LIN {X 0,Y 305.398,Z 312.447,A -85,B 0,C 180,E1 -15799.883,E2 -15799.883} C_VEL
LIN {X 0,Y 305.449,Z 312.421,A -85,B 0,C 180,E1 -15803.636,E2 -15803.636} C_VEL
LIN {X 0,Y 305.452,Z 312.437,A -85,B 0,C 180,E1 -15806.482,E2 -15806.482} C_VEL
LIN {X 0,Y 305.417,Z 312.439,A -85,B 0,C 180,E1 -15809.586,E2 -15809.586} C_VEL
LIN {X 0,Y 305.444,Z 312.436,A -85,B 0,C 180,E1 -15812.601,E2 -15812.601} C_VEL
LIN {X 0,Y 305.461,Z 312.428,A -85,B 0,C 180,E1 -15815.535,E2 -15815.535} C_VEL
LIN {X 0,Y 305.498,Z 312.423,A -85,B 0,C 180,E1 -15819.814,E2 -15819.814} C_VEL
LIN {X 0,Y 305.56,Z 312.415,A -85,B 0,C 180,E1 -15822.602,E2 -15822.602} C_VEL
LIN {X 0,Y 305.635,Z 312.412,A -85,B 0,C 180,E1 -15825.349,E2 -15825.349} C_VEL
LIN {X 0,Y 305.622,Z 312.411,A -85,B 0,C 180,E1 -15829.399,E2 -15829.399} C_VEL
LIN {X 0,Y 305.737,Z 312.393,A -85,B 0,C 180,E1 -15832.073,E2 -15832.073} C_VEL
LIN {X 0,Y 305.66,Z 312.409,A -85,B 0,C 180,E1 -15834.723,E2 -15834.723} C_VEL
LIN {X 0,Y 305.943,Z 312.363,A -85,B 0,C 180,E1 -15838.684,E2 -15838.684} C_VEL
LIN {X 0,Y 305.945,Z 312.371,A -85,B 0,C 180,E1 -15841.317,E2 -15841.317} C_VEL
LIN {X 0,Y 305.838,Z 312.386,A -85,B 0,C 180,E1 -15846.598,E2 -15846.598} C_VEL
LIN {X 0,Y 305.723,Z 312.392,A -85,B 0,C 180,E1 -15849.26,E2 -15849.26} C_VEL
LIN {X 0,Y 305.576,Z 312.407,A -85,B 0,C 180,E1 -15853.297,E2 -15853.297} C_VEL
LIN {X 0,Y 305.581,Z 312.419,A -85,B 0,C 180,E1 -15856.021,E2 -15856.021} C_VEL
LIN {X 0,Y 305.565,Z 312.413,A -85,B 0,C 180,E1 -15859.446,E2 -15859.446} C_VEL
LIN {X 0,Y 305.478,Z 312.424,A -85,B 0,C 180,E1 -15863.042,E2 -15863.042} C_VEL
LIN {X 0,Y 305.543,Z 312.424,A -85,B 0,C 180,E1 -15866.231,E2 -15866.231} C_VEL
LIN {X 0,Y 305.485,Z 312.426,A -85,B 0,C 180,E1 -15869.052,E2 -15869.052} C_VEL
LIN {X 0,Y 305.437,Z 312.43,A -85,B 0,C 180,E1 -15871.953,E2 -15871.953} C_VEL
LIN {X 0,Y 305.453,Z 312.435,A -85,B 0,C 180,E1 -15875.115,E2 -15875.115} C_VEL
LIN {X 0,Y 305.483,Z 312.433,A -85,B 0,C 180,E1 -15878.541,E2 -15878.541} C_VEL
LIN {X 0,Y 305.49,Z 312.429,A -85,B 0,C 180,E1 -15882.597,E2 -15882.597} C_VEL
LIN {X 0,Y 305.485,Z 312.416,A -85,B 0,C 180,E1 -15886.359,E2 -15886.359} C_VEL
LIN {X 0,Y 305.494,Z 312.42,A -85,B 0,C 180,E1 -15889.901,E2 -15889.901} C_VEL
LIN {X 0,Y 305.495,Z 312.51,A -85,B 0,C 180,E1 -15893.574,E2 -15893.574} C_VEL
LIN {X 0,Y 308.431,Z 323.615,A -85,B 0,C 180,E1 -15897.469,E2 -15897.469} C_VEL
LIN {X 0,Y 310.794,Z 334.247,A -85,B 0,C 180,E1 -15900.913,E2 -15900.913} C_VEL
LIN {X 0,Y 311.289,Z 336.675,A -85,B 0,C 180,E1 -15901.649,E2 -15901.649} C_VEL
LIN {X 0,Y 314.76,Z 344.965,A -85,B 0,C 180,E1 -15902.279,E2 -15902.279} C_VEL
LIN {X 0,Y 319.961,Z 370.288,A -85,B 0,C 180,E1 -15903.522,E2 -15903.522} C_VEL
LIN {X 0,Y 321.701,Z 382.338,A -85,B 0,C 180,E1 -15904.017,E2 -15904.017} C_VEL
LIN {X 0,Y 319.792,Z 446.05,A -85,B 0,C 180,E1 -15905.495,E2 -15905.495} C_VEL
LIN {X 0,Y 318.807,Z 458.991,A -85,B 0,C 180,E1 -15906.02,E2 -15906.02} C_VEL
LIN {X 0,Y 317.343,Z 471.558,A -85,B 0,C 180,E1 -15906.769,E2 -15906.769} C_VEL
LIN {X 0,Y 315.685,Z 483.551,A -85,B 0,C 180,E1 -15907.764,E2 -15907.764} C_VEL
LIN {X 0,Y 313.762,Z 495.004,A -85,B 0,C 180,E1 -15909.001,E2 -15909.001} C_VEL
LIN {X 0,Y 311.866,Z 505.349,A -85,B 0,C 180,E1 -15910.417,E2 -15910.417} C_VEL
LIN {X 0,Y 310.092,Z 513.837,A -85,B 0,C 180,E1 -15911.845,E2 -15911.845} C_VEL
LIN {X 0,Y 308.629,Z 521.845,A -85,B 0,C 180,E1 -15913.503,E2 -15913.503} C_VEL
LIN {X 0,Y 307.051,Z 529.381,A -85,B 0,C 180,E1 -15915.42,E2 -15915.42} C_VEL
LIN {X 0,Y 305.65,Z 535.589,A -85,B 0,C 180,E1 -15917.385,E2 -15917.385} C_VEL
LIN {X 0,Y 304.733,Z 540.548,A -85,B 0,C 180,E1 -15919.37,E2 -15919.37} C_VEL
LIN {X 0,Y 304.146,Z 544.402,A -85,B 0,C 180,E1 -15921.364,E2 -15921.364} C_VEL
LIN {X 0,Y 303.744,Z 547.251,A -85,B 0,C 180,E1 -15923.359,E2 -15923.359} C_VEL
LIN {X 0,Y 303.632,Z 549.583,A -85,B 0,C 180,E1 -15926.02,E2 -15926.02} C_VEL
LIN {X 0,Y 303.623,Z 550.168,A -85,B 0,C 180,E1 -15927.349,E2 -15927.349} C_VEL
LIN {X 0,Y 303.607,Z 550.324,A -85,B 0,C 180,E1 -15928.676,E2 -15928.676} C_VEL
LIN {X 0,Y 303.67,Z 550.08,A -85,B 0,C 180,E1 -15930.002,E2 -15930.002} C_VEL
LIN {X 0,Y 303.636,Z 549.443,A -85,B 0,C 180,E1 -15931.328,E2 -15931.328} C_VEL
LIN {X 0,Y 303.646,Z 548.413,A -85,B 0,C 180,E1 -15932.655,E2 -15932.655} C_VEL
LIN {X 0,Y 303.671,Z 546.934,A -85,B 0,C 180,E1 -15933.983,E2 -15933.983} C_VEL
LIN {X 0,Y 303.732,Z 544.307,A -85,B 0,C 180,E1 -15935.746,E2 -15935.746} C_VEL
LIN {X 0,Y 303.942,Z 539.784,A -85,B 0,C 180,E1 -15937.977,E2 -15937.977} C_VEL
LIN {X 0,Y 304.442,Z 533.453,A -85,B 0,C 180,E1 -15940.308,E2 -15940.308} C_VEL
LIN {X 0,Y 305.118,Z 526.541,A -85,B 0,C 180,E1 -15942.304,E2 -15942.304} C_VEL
LIN {X 0,Y 305.993,Z 519.484,A -85,B 0,C 180,E1 -15943.957,E2 -15943.957} C_VEL
LIN {X 0,Y 307.039,Z 510.967,A -85,B 0,C 180,E1 -15945.604,E2 -15945.604} C_VEL
LIN {X 0,Y 308.259,Z 500.414,A -85,B 0,C 180,E1 -15947.243,E2 -15947.243} C_VEL
LIN {X 0,Y 309.206,Z 491.39,A -85,B 0,C 180,E1 -15948.385,E2 -15948.385} C_VEL
LIN {X 0,Y 310.42,Z 480.275,A -85,B 0,C 180,E1 -15949.51,E2 -15949.51} C_VEL
LIN {X 0,Y 311.558,Z 467.945,A -85,B 0,C 180,E1 -15950.467,E2 -15950.467} C_VEL
LIN {X 0,Y 312.492,Z 454.939,A -85,B 0,C 180,E1 -15951.179,E2 -15951.179} C_VEL
LIN {X 0,Y 313.069,Z 441.053,A -85,B 0,C 180,E1 -15951.656,E2 -15951.656} C_VEL
LIN {X 0,Y 314.281,Z 379.106,A -85,B 0,C 180,E1 -15953.068,E2 -15953.068} C_VEL
LIN {X 0,Y 308.709,Z 337.55,A -85,B 0,C 180,E1 -15954.454,E2 -15954.454} C_VEL
LIN {X 0,Y 309.301,Z 331.86,A -85,B 0,C 180,E1 -15955.94,E2 -15955.94} C_VEL
LIN {X 0,Y 307.601,Z 322.197,A -85,B 0,C 180,E1 -15958.674,E2 -15958.674} C_VEL
LIN {X 0,Y 305.475,Z 312.435,A -85,B 0,C 180,E1 -15961.581,E2 -15961.581} C_VEL
LIN {X 0,Y 305.469,Z 312.433,A -85,B 0,C 180,E1 -15965.114,E2 -15965.114} C_VEL
LIN {X 0,Y 305.456,Z 312.438,A -85,B 0,C 180,E1 -15968.53,E2 -15968.53} C_VEL
LIN {X 0,Y 305.462,Z 312.438,A -85,B 0,C 180,E1 -15972.587,E2 -15972.587} C_VEL
LIN {X 0,Y 305.432,Z 312.439,A -85,B 0,C 180,E1 -15976.346,E2 -15976.346} C_VEL
LIN {X 0,Y 305.465,Z 312.431,A -85,B 0,C 180,E1 -15979.893,E2 -15979.893} C_VEL
LIN {X 0,Y 305.487,Z 312.429,A -85,B 0,C 180,E1 -15983.632,E2 -15983.632} C_VEL
LIN {X 0,Y 305.472,Z 312.431,A -85,B 0,C 180,E1 -15986.484,E2 -15986.484} C_VEL
LIN {X 0,Y 305.503,Z 312.429,A -85,B 0,C 180,E1 -15990.951,E2 -15990.951} C_VEL
LIN {X 0,Y 305.579,Z 312.418,A -85,B 0,C 180,E1 -15994.088,E2 -15994.088} C_VEL
LIN {X 0,Y 305.481,Z 312.429,A -85,B 0,C 180,E1 -15998.401,E2 -15998.401} C_VEL
LIN {X 0,Y 305.525,Z 312.424,A -85,B 0,C 180,E1 -16001.213,E2 -16001.213} C_VEL
LIN {X 0,Y 305.633,Z 312.412,A -85,B 0,C 180,E1 -16005.348,E2 -16005.348} C_VEL
LIN {X 0,Y 305.642,Z 312.412,A -85,B 0,C 180,E1 -16009.4,E2 -16009.4} C_VEL
LIN {X 0,Y 305.754,Z 312.392,A -85,B 0,C 180,E1 -16012.072,E2 -16012.072} C_VEL
LIN {X 0,Y 305.677,Z 312.401,A -85,B 0,C 180,E1 -16014.723,E2 -16014.723} C_VEL
LIN {X 0,Y 305.96,Z 312.37,A -85,B 0,C 180,E1 -16018.683,E2 -16018.683} C_VEL
LIN {X 0,Y 305.96,Z 312.369,A -85,B 0,C 180,E1 -16021.316,E2 -16021.316} C_VEL
LIN {X 0,Y 305.687,Z 312.396,A -85,B 0,C 180,E1 -16025.276,E2 -16025.276} C_VEL
LIN {X 0,Y 305.778,Z 312.389,A -85,B 0,C 180,E1 -16027.926,E2 -16027.926} C_VEL
LIN {X 0,Y 305.605,Z 312.415,A -85,B 0,C 180,E1 -16031.945,E2 -16031.945} C_VEL
LIN {X 0,Y 305.615,Z 312.413,A -85,B 0,C 180,E1 -16035.014,E2 -16035.014} C_VEL
LIN {X 0,Y 305.524,Z 312.43,A -85,B 0,C 180,E1 -16038.786,E2 -16038.786} C_VEL
LIN {X 0,Y 305.492,Z 312.432,A -85,B 0,C 180,E1 -16043.039,E2 -16043.039} C_VEL
LIN {X 0,Y 305.532,Z 312.423,A -85,B 0,C 180,E1 -16046.218,E2 -16046.218} C_VEL
LIN {X 0,Y 305.494,Z 312.431,A -85,B 0,C 180,E1 -16049.047,E2 -16049.047} C_VEL
LIN {X 0,Y 305.448,Z 312.433,A -85,B 0,C 180,E1 -16051.951,E2 -16051.951} C_VEL
LIN {X 0,Y 305.468,Z 312.434,A -85,B 0,C 180,E1 -16055.112,E2 -16055.112} C_VEL
LIN {X 0,Y 305.445,Z 312.433,A -85,B 0,C 180,E1 -16058.525,E2 -16058.525} C_VEL
LIN {X 0,Y 305.478,Z 312.429,A -85,B 0,C 180,E1 -16062.588,E2 -16062.588} C_VEL
LIN {X 0,Y 305.459,Z 312.435,A -85,B 0,C 180,E1 -16067.413,E2 -16067.413} C_VEL
LIN {X 0,Y 305.499,Z 312.43,A -85,B 0,C 180,E1 -16071.599,E2 -16071.599} C_VEL
LIN {X 0,Y 305.466,Z 312.431,A -85,B 0,C 180,E1 -16074.885,E2 -16074.885} C_VEL
LIN {X 0,Y 305.453,Z 312.435,A -85,B 0,C 180,E1 -16078.354,E2 -16078.354} C_VEL
LIN {X 0,Y 305.516,Z 312.425,A -85,B 0,C 180,E1 -16081.112,E2 -16081.112} C_VEL
LIN {X 0,Y 305.574,Z 312.423,A -85,B 0,C 180,E1 -16084.086,E2 -16084.086} C_VEL
LIN {X 0,Y 305.532,Z 312.428,A -85,B 0,C 180,E1 -16088.403,E2 -16088.403} C_VEL
LIN {X 0,Y 305.595,Z 312.416,A -85,B 0,C 180,E1 -16091.216,E2 -16091.216} C_VEL
LIN {X 0,Y 305.651,Z 312.41,A -85,B 0,C 180,E1 -16095.347,E2 -16095.347} C_VEL
LIN {X 0,Y 305.665,Z 312.589,A -85,B 0,C 180,E1 -16099.231,E2 -16099.231} C_VEL
LIN {X 0,Y 306.522,Z 316.593,A -85,B 0,C 180,E1 -16100.487,E2 -16100.487} C_VEL
LIN {X 0,Y 312.904,Z 335.521,A -85,B 0,C 180,E1 -16101.395,E2 -16101.395} C_VEL
LIN {X 0,Y 314.899,Z 346.476,A -85,B 0,C 180,E1 -16101.787,E2 -16101.787} C_VEL
LIN {X 0,Y 313.086,Z 424.785,A -85,B 0,C 180,E1 -16103.594,E2 -16103.594} C_VEL
LIN {X 0,Y 312.418,Z 438.468,A -85,B 0,C 180,E1 -16104.188,E2 -16104.188} C_VEL
LIN {X 0,Y 311.682,Z 450.742,A -85,B 0,C 180,E1 -16104.985,E2 -16104.985} C_VEL
LIN {X 0,Y 310.637,Z 463.358,A -85,B 0,C 180,E1 -16106.106,E2 -16106.106} C_VEL
LIN {X 0,Y 309.466,Z 474.611,A -85,B 0,C 180,E1 -16107.395,E2 -16107.395} C_VEL
LIN {X 0,Y 308.216,Z 484.757,A -85,B 0,C 180,E1 -16108.855,E2 -16108.855} C_VEL
LIN {X 0,Y 306.982,Z 494.708,A -85,B 0,C 180,E1 -16110.654,E2 -16110.654} C_VEL
LIN {X 0,Y 305.871,Z 503.471,A -85,B 0,C 180,E1 -16112.632,E2 -16112.632} C_VEL
LIN {X 0,Y 305.06,Z 510.446,A -85,B 0,C 180,E1 -16114.623,E2 -16114.623} C_VEL
LIN {X 0,Y 304.552,Z 516.023,A -85,B 0,C 180,E1 -16116.624,E2 -16116.624} C_VEL
LIN {X 0,Y 304.078,Z 520.42,A -85,B 0,C 180,E1 -16118.638,E2 -16118.638} C_VEL
LIN {X 0,Y 303.697,Z 523.738,A -85,B 0,C 180,E1 -16120.667,E2 -16120.667} C_VEL
LIN {X 0,Y 303.593,Z 525.384,A -85,B 0,C 180,E1 -16122.023,E2 -16122.023} C_VEL
LIN {X 0,Y 303.543,Z 526.681,A -85,B 0,C 180,E1 -16123.485,E2 -16123.485} C_VEL
LIN {X 0,Y 303.461,Z 527.755,A -85,B 0,C 180,E1 -16126.133,E2 -16126.133} C_VEL
LIN {X 0,Y 303.688,Z 527.448,A -85,B 0,C 180,E1 -16128.409,E2 -16128.409} C_VEL
LIN {X 0,Y 303.99,Z 526.316,A -85,B 0,C 180,E1 -16130.289,E2 -16130.289} C_VEL
LIN {X 0,Y 304.616,Z 523.753,A -85,B 0,C 180,E1 -16132.652,E2 -16132.652} C_VEL
LIN {X 0,Y 305.608,Z 519.497,A -85,B 0,C 180,E1 -16135.176,E2 -16135.176} C_VEL
LIN {X 0,Y 306.708,Z 514.599,A -85,B 0,C 180,E1 -16137.274,E2 -16137.274} C_VEL
LIN {X 0,Y 308.159,Z 508.31,A -85,B 0,C 180,E1 -16139.36,E2 -16139.36} C_VEL
LIN {X 0,Y 309.903,Z 500.374,A -85,B 0,C 180,E1 -16141.437,E2 -16141.437} C_VEL
LIN {X 0,Y 311.708,Z 491.871,A -85,B 0,C 180,E1 -16143.192,E2 -16143.192} C_VEL
LIN {X 0,Y 313.595,Z 481.907,A -85,B 0,C 180,E1 -16144.851,E2 -16144.851} C_VEL
LIN {X 0,Y 315.375,Z 471.812,A -85,B 0,C 180,E1 -16146.192,E2 -16146.192} C_VEL
LIN {X 0,Y 316.932,Z 461.289,A -85,B 0,C 180,E1 -16147.313,E2 -16147.313} C_VEL
LIN {X 0,Y 318.315,Z 449.539,A -85,B 0,C 180,E1 -16148.283,E2 -16148.283} C_VEL
LIN {X 0,Y 319.552,Z 436.467,A -85,B 0,C 180,E1 -16149.065,E2 -16149.065} C_VEL
LIN {X 0,Y 320.342,Z 423.599,A -85,B 0,C 180,E1 -16149.575,E2 -16149.575} C_VEL
LIN {X 0,Y 322.577,Z 350.795,A -85,B 0,C 180,E1 -16151.238,E2 -16151.238} C_VEL
LIN {X 0,Y 316.186,Z 336.137,A -85,B 0,C 180,E1 -16152.328,E2 -16152.328} C_VEL
LIN {X 0,Y 308.719,Z 321.185,A -85,B 0,C 180,E1 -16153.627,E2 -16153.627} C_VEL
LIN {X 0,Y 306.652,Z 317.269,A -85,B 0,C 180,E1 -16154.031,E2 -16154.031} C_VEL
LIN {X 0,Y 305.411,Z 312.433,A -85,B 0,C 180,E1 -16155.821,E2 -16155.821} C_VEL
LIN {X 0,Y 305.404,Z 312.433,A -85,B 0,C 180,E1 -16156.566,E2 -16156.566} C_VEL
LIN {X 0,Y 304.731,Z 312.527,A -85,B 0,C 180,E1 -16157.666,E2 -16157.666} C_VEL
LIN {X 0,Y 301.878,Z 312.895,A -85,B 0,C 180,E1 -16159.458,E2 -16159.458} C_VEL
LIN {X 0,Y 299.471,Z 313.197,A -85,B 0,C 180,E1 -16160.912,E2 -16160.912} C_VEL
LIN {X 0,Y 298.452,Z 313.314,A -85,B 0,C 180,E1 -16162.038,E2 -16162.038} C_VEL
LIN {X 0,Y 298.375,Z 313.318,A -85,B 0,C 180,E1 -16162.419,E2 -16162.419} C_VEL
LIN {X 0,Y 298.395,Z 313.301,A -85,B 0,C 180,E1 -16165.58,E2 -16165.58} C_VEL
LIN {X 0,Y 298.364,Z 313.313,A -85,B 0,C 180,E1 -16168.788,E2 -16168.788} C_VEL
LIN {X 0,Y 298.4,Z 313.309,A -85,B 0,C 180,E1 -16171.898,E2 -16171.898} C_VEL
LIN {X 0,Y 298.426,Z 313.304,A -85,B 0,C 180,E1 -16174.919,E2 -16174.919} C_VEL
LIN {X 0,Y 298.426,Z 313.301,A -85,B 0,C 180,E1 -16179.314,E2 -16179.314} C_VEL
LIN {X 0,Y 298.524,Z 313.295,A -85,B 0,C 180,E1 -16182.179,E2 -16182.179} C_VEL
LIN {X 0,Y 298.58,Z 313.291,A -85,B 0,C 180,E1 -16184.994,E2 -16184.994} C_VEL
LIN {X 0,Y 298.578,Z 313.288,A -85,B 0,C 180,E1 -16189.146,E2 -16189.146} C_VEL
LIN {X 0,Y 298.688,Z 313.273,A -85,B 0,C 180,E1 -16191.884,E2 -16191.884} C_VEL
LIN {X 0,Y 298.629,Z 313.283,A -85,B 0,C 180,E1 -16194.599,E2 -16194.599} C_VEL
LIN {X 0,Y 298.91,Z 313.239,A -85,B 0,C 180,E1 -16198.653,E2 -16198.653} C_VEL
LIN {X 0,Y 298.911,Z 313.248,A -85,B 0,C 180,E1 -16201.348,E2 -16201.348} C_VEL
LIN {X 0,Y 298.784,Z 313.263,A -85,B 0,C 180,E1 -16206.754,E2 -16206.754} C_VEL
LIN {X 0,Y 298.668,Z 313.272,A -85,B 0,C 180,E1 -16209.481,E2 -16209.481} C_VEL
LIN {X 0,Y 298.539,Z 313.282,A -85,B 0,C 180,E1 -16213.616,E2 -16213.616} C_VEL
LIN {X 0,Y 298.536,Z 313.298,A -85,B 0,C 180,E1 -16216.41,E2 -16216.41} C_VEL
LIN {X 0,Y 298.5,Z 313.295,A -85,B 0,C 180,E1 -16219.656,E2 -16219.656} C_VEL
LIN {X 0,Y 298.446,Z 313.298,A -85,B 0,C 180,E1 -16223.599,E2 -16223.599} C_VEL
LIN {X 0,Y 298.481,Z 313.305,A -85,B 0,C 180,E1 -16226.576,E2 -16226.576} C_VEL
LIN {X 0,Y 298.411,Z 313.315,A -85,B 0,C 180,E1 -16229.642,E2 -16229.642} C_VEL
LIN {X 0,Y 298.387,Z 313.31,A -85,B 0,C 180,E1 -16232.802,E2 -16232.802} C_VEL
LIN {X 0,Y 298.461,Z 313.306,A -85,B 0,C 180,E1 -16236.816,E2 -16236.816} C_VEL
LIN {X 0,Y 298.411,Z 313.318,A -85,B 0,C 180,E1 -16241.097,E2 -16241.097} C_VEL
LIN {X 0,Y 298.451,Z 313.308,A -85,B 0,C 180,E1 -16243.118,E2 -16243.118} C_VEL
LIN {X 0,Y 298.46,Z 313.295,A -85,B 0,C 180,E1 -16246.934,E2 -16246.934} C_VEL
LIN {X 0,Y 298.434,Z 313.303,A -85,B 0,C 180,E1 -16251,E2 -16251} C_VEL
LIN {X 0,Y 298.444,Z 313.405,A -85,B 0,C 180,E1 -16252.779,E2 -16252.779} C_VEL
LIN {X 0,Y 300.953,Z 322.896,A -85,B 0,C 180,E1 -16256.255,E2 -16256.255} C_VEL
LIN {X 0,Y 303.087,Z 331.928,A -85,B 0,C 180,E1 -16259.33,E2 -16259.33} C_VEL
LIN {X 0,Y 304.092,Z 336.451,A -85,B 0,C 180,E1 -16260.755,E2 -16260.755} C_VEL
LIN {X 0,Y 309.003,Z 347.527,A -85,B 0,C 180,E1 -16261.672,E2 -16261.672} C_VEL
LIN {X 0,Y 313.784,Z 371.061,A -85,B 0,C 180,E1 -16262.866,E2 -16262.866} C_VEL
LIN {X 0,Y 315.584,Z 382.767,A -85,B 0,C 180,E1 -16263.375,E2 -16263.375} C_VEL
LIN {X 0,Y 313.624,Z 445.356,A -85,B 0,C 180,E1 -16264.847,E2 -16264.847} C_VEL
LIN {X 0,Y 312.605,Z 458.435,A -85,B 0,C 180,E1 -16265.381,E2 -16265.381} C_VEL
LIN {X 0,Y 311.035,Z 471.63,A -85,B 0,C 180,E1 -16266.181,E2 -16266.181} C_VEL
LIN {X 0,Y 309.432,Z 482.739,A -85,B 0,C 180,E1 -16267.113,E2 -16267.113} C_VEL
LIN {X 0,Y 307.459,Z 494.288,A -85,B 0,C 180,E1 -16268.374,E2 -16268.374} C_VEL
LIN {X 0,Y 305.415,Z 504.707,A -85,B 0,C 180,E1 -16269.81,E2 -16269.81} C_VEL
LIN {X 0,Y 303.315,Z 514.297,A -85,B 0,C 180,E1 -16271.459,E2 -16271.459} C_VEL
LIN {X 0,Y 301.763,Z 522.232,A -85,B 0,C 180,E1 -16273.171,E2 -16273.171} C_VEL
LIN {X 0,Y 300.186,Z 529.458,A -85,B 0,C 180,E1 -16275.079,E2 -16275.079} C_VEL
LIN {X 0,Y 298.72,Z 535.6,A -85,B 0,C 180,E1 -16277.087,E2 -16277.087} C_VEL
LIN {X 0,Y 297.735,Z 540.5,A -85,B 0,C 180,E1 -16279.117,E2 -16279.117} C_VEL
LIN {X 0,Y 297.089,Z 544.298,A -85,B 0,C 180,E1 -16281.157,E2 -16281.157} C_VEL
LIN {X 0,Y 296.69,Z 547.096,A -85,B 0,C 180,E1 -16283.2,E2 -16283.2} C_VEL
LIN {X 0,Y 296.53,Z 549.378,A -85,B 0,C 180,E1 -16285.925,E2 -16285.925} C_VEL
LIN {X 0,Y 296.548,Z 549.929,A -85,B 0,C 180,E1 -16287.285,E2 -16287.285} C_VEL
LIN {X 0,Y 296.582,Z 549.778,A -85,B 0,C 180,E1 -16290.002,E2 -16290.002} C_VEL
LIN {X 0,Y 296.552,Z 549.116,A -85,B 0,C 180,E1 -16291.36,E2 -16291.36} C_VEL
LIN {X 0,Y 296.571,Z 548.055,A -85,B 0,C 180,E1 -16292.719,E2 -16292.719} C_VEL
LIN {X 0,Y 296.587,Z 546.53,A -85,B 0,C 180,E1 -16294.078,E2 -16294.078} C_VEL
LIN {X 0,Y 296.678,Z 543.442,A -85,B 0,C 180,E1 -16296.121,E2 -16296.121} C_VEL
LIN {X 0,Y 296.876,Z 539.267,A -85,B 0,C 180,E1 -16298.168,E2 -16298.168} C_VEL
LIN {X 0,Y 297.411,Z 532.872,A -85,B 0,C 180,E1 -16300.554,E2 -16300.554} C_VEL
LIN {X 0,Y 298.155,Z 525.892,A -85,B 0,C 180,E1 -16302.596,E2 -16302.596} C_VEL
LIN {X 0,Y 299.028,Z 518.75,A -85,B 0,C 180,E1 -16304.289,E2 -16304.289} C_VEL
LIN {X 0,Y 300.143,Z 510.107,A -85,B 0,C 180,E1 -16305.972,E2 -16305.972} C_VEL
LIN {X 0,Y 301.415,Z 499.411,A -85,B 0,C 180,E1 -16307.647,E2 -16307.647} C_VEL
LIN {X 0,Y 302.485,Z 490.242,A -85,B 0,C 180,E1 -16308.808,E2 -16308.808} C_VEL
LIN {X 0,Y 303.695,Z 478.905,A -85,B 0,C 180,E1 -16309.96,E2 -16309.96} C_VEL
LIN {X 0,Y 304.787,Z 467.401,A -85,B 0,C 180,E1 -16310.855,E2 -16310.855} C_VEL
LIN {X 0,Y 305.727,Z 454.228,A -85,B 0,C 180,E1 -16311.582,E2 -16311.582} C_VEL
LIN {X 0,Y 306.284,Z 441.568,A -85,B 0,C 180,E1 -16312.028,E2 -16312.028} C_VEL
LIN {X 0,Y 307.547,Z 379.797,A -85,B 0,C 180,E1 -16313.469,E2 -16313.469} C_VEL
LIN {X 0,Y 301.866,Z 337.34,A -85,B 0,C 180,E1 -16314.912,E2 -16314.912} C_VEL
LIN {X 0,Y 302.275,Z 332.48,A -85,B 0,C 180,E1 -16316.218,E2 -16316.218} C_VEL
LIN {X 0,Y 300.19,Z 321.402,A -85,B 0,C 180,E1 -16319.451,E2 -16319.451} C_VEL
LIN {X 0,Y 298.431,Z 313.308,A -85,B 0,C 180,E1 -16321.956,E2 -16321.956} C_VEL
LIN {X 0,Y 298.425,Z 313.312,A -85,B 0,C 180,E1 -16326.071,E2 -16326.071} C_VEL
LIN {X 0,Y 298.41,Z 313.311,A -85,B 0,C 180,E1 -16329.488,E2 -16329.488} C_VEL
LIN {X 0,Y 298.406,Z 313.313,A -85,B 0,C 180,E1 -16333.104,E2 -16333.104} C_VEL
LIN {X 0,Y 298.41,Z 313.314,A -85,B 0,C 180,E1 -16336.922,E2 -16336.922} C_VEL
LIN {X 0,Y 298.406,Z 313.314,A -85,B 0,C 180,E1 -16341.008,E2 -16341.008} C_VEL
LIN {X 0,Y 298.425,Z 313.308,A -85,B 0,C 180,E1 -16343.931,E2 -16343.931} C_VEL
LIN {X 0,Y 298.402,Z 313.311,A -85,B 0,C 180,E1 -16347.984,E2 -16347.984} C_VEL
LIN {X 0,Y 298.477,Z 313.302,A -85,B 0,C 180,E1 -16351.905,E2 -16351.905} C_VEL
LIN {X 0,Y 298.492,Z 313.303,A -85,B 0,C 180,E1 -16354.924,E2 -16354.924} C_VEL
LIN {X 0,Y 298.43,Z 313.311,A -85,B 0,C 180,E1 -16359.314,E2 -16359.314} C_VEL
LIN {X 0,Y 298.473,Z 313.297,A -85,B 0,C 180,E1 -16362.175,E2 -16362.175} C_VEL
LIN {X 0,Y 298.593,Z 313.287,A -85,B 0,C 180,E1 -16364.994,E2 -16364.994} C_VEL
LIN {X 0,Y 298.598,Z 313.287,A -85,B 0,C 180,E1 -16369.147,E2 -16369.147} C_VEL
LIN {X 0,Y 298.705,Z 313.271,A -85,B 0,C 180,E1 -16371.884,E2 -16371.884} C_VEL
LIN {X 0,Y 298.645,Z 313.276,A -85,B 0,C 180,E1 -16374.598,E2 -16374.598} C_VEL
LIN {X 0,Y 298.927,Z 313.247,A -85,B 0,C 180,E1 -16378.653,E2 -16378.653} C_VEL
LIN {X 0,Y 298.927,Z 313.245,A -85,B 0,C 180,E1 -16381.347,E2 -16381.347} C_VEL
LIN {X 0,Y 298.782,Z 313.26,A -85,B 0,C 180,E1 -16386.754,E2 -16386.754} C_VEL
LIN {X 0,Y 298.632,Z 313.28,A -85,B 0,C 180,E1 -16389.482,E2 -16389.482} C_VEL
LIN {X 0,Y 298.552,Z 313.292,A -85,B 0,C 180,E1 -16393.615,E2 -16393.615} C_VEL
LIN {X 0,Y 298.49,Z 313.301,A -85,B 0,C 180,E1 -16396.412,E2 -16396.412} C_VEL
LIN {X 0,Y 298.466,Z 313.304,A -85,B 0,C 180,E1 -16399.626,E2 -16399.626} C_VEL
LIN {X 0,Y 298.435,Z 313.307,A -85,B 0,C 180,E1 -16403.599,E2 -16403.599} C_VEL
LIN {X 0,Y 298.491,Z 313.302,A -85,B 0,C 180,E1 -16406.574,E2 -16406.574} C_VEL
LIN {X 0,Y 298.422,Z 313.309,A -85,B 0,C 180,E1 -16409.64,E2 -16409.64} C_VEL
LIN {X 0,Y 298.4,Z 313.313,A -85,B 0,C 180,E1 -16412.799,E2 -16412.799} C_VEL
LIN {X 0,Y 298.45,Z 313.306,A -85,B 0,C 180,E1 -16416.806,E2 -16416.806} C_VEL
LIN {X 0,Y 298.417,Z 313.31,A -85,B 0,C 180,E1 -16421.256,E2 -16421.256} C_VEL
LIN {X 0,Y 298.359,Z 313.317,A -85,B 0,C 180,E1 -16425.034,E2 -16425.034} C_VEL
LIN {X 0,Y 298.389,Z 313.313,A -85,B 0,C 180,E1 -16428.737,E2 -16428.737} C_VEL
LIN {X 0,Y 298.429,Z 313.31,A -85,B 0,C 180,E1 -16432.242,E2 -16432.242} C_VEL
LIN {X 0,Y 298.412,Z 313.312,A -85,B 0,C 180,E1 -16435.58,E2 -16435.58} C_VEL
LIN {X 0,Y 298.395,Z 313.312,A -85,B 0,C 180,E1 -16438.789,E2 -16438.789} C_VEL
LIN {X 0,Y 298.462,Z 313.308,A -85,B 0,C 180,E1 -16441.902,E2 -16441.902} C_VEL
LIN {X 0,Y 298.489,Z 313.302,A -85,B 0,C 180,E1 -16444.922,E2 -16444.922} C_VEL
LIN {X 0,Y 298.468,Z 313.303,A -85,B 0,C 180,E1 -16449.315,E2 -16449.315} C_VEL
LIN {X 0,Y 298.542,Z 313.298,A -85,B 0,C 180,E1 -16452.178,E2 -16452.178} C_VEL
LIN {X 0,Y 298.596,Z 313.291,A -85,B 0,C 180,E1 -16454.993,E2 -16454.993} C_VEL
LIN {X 0,Y 298.619,Z 313.431,A -85,B 0,C 180,E1 -16458.888,E2 -16458.888} C_VEL
LIN {X 0,Y 299.331,Z 316.889,A -85,B 0,C 180,E1 -16459.994,E2 -16459.994} C_VEL
LIN {X 0,Y 306.12,Z 336.457,A -85,B 0,C 180,E1 -16460.969,E2 -16460.969} C_VEL
LIN {X 0,Y 308.206,Z 347.657,A -85,B 0,C 180,E1 -16461.383,E2 -16461.383} C_VEL
LIN {X 0,Y 306.322,Z 424.841,A -85,B 0,C 180,E1 -16463.197,E2 -16463.197} C_VEL
LIN {X 0,Y 305.623,Z 438.713,A -85,B 0,C 180,E1 -16463.81,E2 -16463.81} C_VEL
LIN {X 0,Y 304.865,Z 450.988,A -85,B 0,C 180,E1 -16464.624,E2 -16464.624} C_VEL
LIN {X 0,Y 303.845,Z 462.823,A -85,B 0,C 180,E1 -16465.687,E2 -16465.687} C_VEL
LIN {X 0,Y 302.601,Z 474.656,A -85,B 0,C 180,E1 -16467.059,E2 -16467.059} C_VEL
LIN {X 0,Y 301.377,Z 484.506,A -85,B 0,C 180,E1 -16468.495,E2 -16468.495} C_VEL
LIN {X 0,Y 300.08,Z 494.552,A -85,B 0,C 180,E1 -16470.333,E2 -16470.333} C_VEL
LIN {X 0,Y 298.909,Z 503.396,A -85,B 0,C 180,E1 -16472.356,E2 -16472.356} C_VEL
LIN {X 0,Y 298.054,Z 510.45,A -85,B 0,C 180,E1 -16474.393,E2 -16474.393} C_VEL
LIN {X 0,Y 297.434,Z 516.895,A -85,B 0,C 180,E1 -16476.783,E2 -16476.783} C_VEL
LIN {X 0,Y 296.946,Z 521.158,A -85,B 0,C 180,E1 -16478.847,E2 -16478.847} C_VEL
LIN {X 0,Y 296.568,Z 524.346,A -85,B 0,C 180,E1 -16480.926,E2 -16480.926} C_VEL
LIN {X 0,Y 296.474,Z 525.928,A -85,B 0,C 180,E1 -16482.316,E2 -16482.316} C_VEL
LIN {X 0,Y 296.435,Z 527.043,A -85,B 0,C 180,E1 -16483.712,E2 -16483.712} C_VEL
LIN {X 0,Y 296.351,Z 527.751,A -85,B 0,C 180,E1 -16485.119,E2 -16485.119} C_VEL
LIN {X 0,Y 296.384,Z 528.058,A -85,B 0,C 180,E1 -16486.53,E2 -16486.53} C_VEL
LIN {X 0,Y 296.617,Z 527.713,A -85,B 0,C 180,E1 -16488.603,E2 -16488.603} C_VEL
LIN {X 0,Y 297.001,Z 526.369,A -85,B 0,C 180,E1 -16490.788,E2 -16490.788} C_VEL
LIN {X 0,Y 297.632,Z 524.016,A -85,B 0,C 180,E1 -16492.941,E2 -16492.941} C_VEL
LIN {X 0,Y 298.468,Z 520.615,A -85,B 0,C 180,E1 -16495.075,E2 -16495.075} C_VEL
LIN {X 0,Y 299.631,Z 515.912,A -85,B 0,C 180,E1 -16497.26,E2 -16497.26} C_VEL
LIN {X 0,Y 301.283,Z 509.019,A -85,B 0,C 180,E1 -16499.666,E2 -16499.666} C_VEL
LIN {X 0,Y 303.163,Z 501.023,A -85,B 0,C 180,E1 -16501.827,E2 -16501.827} C_VEL
LIN {X 0,Y 304.986,Z 492.88,A -85,B 0,C 180,E1 -16503.574,E2 -16503.574} C_VEL
LIN {X 0,Y 307.009,Z 482.776,A -85,B 0,C 180,E1 -16505.308,E2 -16505.308} C_VEL
LIN {X 0,Y 309.022,Z 471.915,A -85,B 0,C 180,E1 -16506.786,E2 -16506.786} C_VEL
LIN {X 0,Y 310.813,Z 460.145,A -85,B 0,C 180,E1 -16508.034,E2 -16508.034} C_VEL
LIN {X 0,Y 312.346,Z 447.529,A -85,B 0,C 180,E1 -16509.049,E2 -16509.049} C_VEL
LIN {X 0,Y 313.513,Z 435.247,A -85,B 0,C 180,E1 -16509.758,E2 -16509.758} C_VEL
LIN {X 0,Y 314.217,Z 423.023,A -85,B 0,C 180,E1 -16510.225,E2 -16510.225} C_VEL
LIN {X 0,Y 316.441,Z 352.704,A -85,B 0,C 180,E1 -16511.859,E2 -16511.859} C_VEL
LIN {X 0,Y 309.928,Z 337.795,A -85,B 0,C 180,E1 -16513.019,E2 -16513.019} C_VEL
LIN {X 0,Y 302.923,Z 324.164,A -85,B 0,C 180,E1 -16514.279,E2 -16514.279} C_VEL
LIN {X 0,Y 299.517,Z 317.579,A -85,B 0,C 180,E1 -16514.962,E2 -16514.962} C_VEL
LIN {X 0,Y 298.373,Z 313.309,A -85,B 0,C 180,E1 -16516.604,E2 -16516.604} C_VEL
LIN {X 0,Y 298.373,Z 313.318,A -85,B 0,C 180,E1 -16521.01,E2 -16521.01} C_VEL
LIN {X 0,Y 298.375,Z 313.318,A -85,B 0,C 180,E1 -16522.419,E2 -16522.419} C_VEL
LIN {X 0,Y 297.733,Z 313.384,A -85,B 0,C 180,E1 -16523.546,E2 -16523.546} C_VEL
LIN {X 0,Y 294.912,Z 313.736,A -85,B 0,C 180,E1 -16525.382,E2 -16525.382} C_VEL
LIN {X 0,Y 292.487,Z 314.053,A -85,B 0,C 180,E1 -16526.872,E2 -16526.872} C_VEL
LIN {X 0,Y 291.418,Z 314.181,A -85,B 0,C 180,E1 -16528.025,E2 -16528.025} C_VEL
LIN {X 0,Y 291.316,Z 314.192,A -85,B 0,C 180,E1 -16528.416,E2 -16528.416} C_VEL
LIN {X 0,Y 291.331,Z 314.192,A -85,B 0,C 180,E1 -16531.153,E2 -16531.153} C_VEL
LIN {X 0,Y 291.346,Z 314.19,A -85,B 0,C 180,E1 -16534.266,E2 -16534.266} C_VEL
LIN {X 0,Y 291.359,Z 314.192,A -85,B 0,C 180,E1 -16537.298,E2 -16537.298} C_VEL
LIN {X 0,Y 291.445,Z 314.177,A -85,B 0,C 180,E1 -16540.27,E2 -16540.27} C_VEL
LIN {X 0,Y 291.542,Z 314.165,A -85,B 0,C 180,E1 -16544.623,E2 -16544.623} C_VEL
LIN {X 0,Y 291.522,Z 314.164,A -85,B 0,C 180,E1 -16548.88,E2 -16548.88} C_VEL
LIN {X 0,Y 291.641,Z 314.153,A -85,B 0,C 180,E1 -16551.687,E2 -16551.687} C_VEL
LIN {X 0,Y 291.597,Z 314.156,A -85,B 0,C 180,E1 -16554.468,E2 -16554.468} C_VEL
LIN {X 0,Y 291.876,Z 314.114,A -85,B 0,C 180,E1 -16558.621,E2 -16558.621} C_VEL
LIN {X 0,Y 291.877,Z 314.124,A -85,B 0,C 180,E1 -16561.38,E2 -16561.38} C_VEL
LIN {X 0,Y 291.733,Z 314.14,A -85,B 0,C 180,E1 -16566.919,E2 -16566.919} C_VEL
LIN {X 0,Y 291.617,Z 314.152,A -85,B 0,C 180,E1 -16569.713,E2 -16569.713} C_VEL
LIN {X 0,Y 291.509,Z 314.157,A -85,B 0,C 180,E1 -16573.951,E2 -16573.951} C_VEL
LIN {X 0,Y 291.475,Z 314.177,A -85,B 0,C 180,E1 -16576.819,E2 -16576.819} C_VEL
LIN {X 0,Y 291.439,Z 314.176,A -85,B 0,C 180,E1 -16579.876,E2 -16579.876} C_VEL
LIN {X 0,Y 291.389,Z 314.178,A -85,B 0,C 180,E1 -16584.207,E2 -16584.207} C_VEL
LIN {X 0,Y 291.415,Z 314.177,A -85,B 0,C 180,E1 -16587.273,E2 -16587.273} C_VEL
LIN {X 0,Y 291.329,Z 314.196,A -85,B 0,C 180,E1 -16590.438,E2 -16590.438} C_VEL
LIN {X 0,Y 291.336,Z 314.198,A -85,B 0,C 180,E1 -16593.7,E2 -16593.7} C_VEL
LIN {X 0,Y 291.396,Z 314.19,A -85,B 0,C 180,E1 -16597.263,E2 -16597.263} C_VEL
LIN {X 0,Y 291.37,Z 314.193,A -85,B 0,C 180,E1 -16600.637,E2 -16600.637} C_VEL
LIN {X 0,Y 291.346,Z 314.189,A -85,B 0,C 180,E1 -16604.392,E2 -16604.392} C_VEL
LIN {X 0,Y 291.383,Z 314.19,A -85,B 0,C 180,E1 -16608.392,E2 -16608.392} C_VEL
LIN {X 0,Y 291.389,Z 314.233,A -85,B 0,C 180,E1 -16611.911,E2 -16611.911} C_VEL
LIN {X 0,Y 293.832,Z 323.35,A -85,B 0,C 180,E1 -16615.388,E2 -16615.388} C_VEL
LIN {X 0,Y 295.953,Z 332.145,A -85,B 0,C 180,E1 -16618.507,E2 -16618.507} C_VEL
LIN {X 0,Y 296.825,Z 335.954,A -85,B 0,C 180,E1 -16619.79,E2 -16619.79} C_VEL
LIN {X 0,Y 303.386,Z 350.423,A -85,B 0,C 180,E1 -16621.063,E2 -16621.063} C_VEL
LIN {X 0,Y 308.09,Z 374.171,A -85,B 0,C 180,E1 -16622.296,E2 -16622.296} C_VEL
LIN {X 0,Y 309.49,Z 384.423,A -85,B 0,C 180,E1 -16622.739,E2 -16622.739} C_VEL
LIN {X 0,Y 307.439,Z 445.741,A -85,B 0,C 180,E1 -16624.213,E2 -16624.213} C_VEL
LIN {X 0,Y 306.313,Z 459.379,A -85,B 0,C 180,E1 -16624.795,E2 -16624.795} C_VEL
LIN {X 0,Y 304.76,Z 471.69,A -85,B 0,C 180,E1 -16625.568,E2 -16625.568} C_VEL
LIN {X 0,Y 302.944,Z 483.498,A -85,B 0,C 180,E1 -16626.594,E2 -16626.594} C_VEL
LIN {X 0,Y 300.907,Z 494.86,A -85,B 0,C 180,E1 -16627.878,E2 -16627.878} C_VEL
LIN {X 0,Y 298.79,Z 505.136,A -85,B 0,C 180,E1 -16629.342,E2 -16629.342} C_VEL
LIN {X 0,Y 296.637,Z 514.401,A -85,B 0,C 180,E1 -16630.99,E2 -16630.99} C_VEL
LIN {X 0,Y 294.902,Z 522.63,A -85,B 0,C 180,E1 -16632.827,E2 -16632.827} C_VEL
LIN {X 0,Y 293.337,Z 529.555,A -85,B 0,C 180,E1 -16634.722,E2 -16634.722} C_VEL
LIN {X 0,Y 291.774,Z 535.626,A -85,B 0,C 180,E1 -16636.774,E2 -16636.774} C_VEL
LIN {X 0,Y 290.751,Z 540.46,A -85,B 0,C 180,E1 -16638.852,E2 -16638.852} C_VEL
LIN {X 0,Y 290.052,Z 544.198,A -85,B 0,C 180,E1 -16640.941,E2 -16640.941} C_VEL
LIN {X 0,Y 289.608,Z 546.941,A -85,B 0,C 180,E1 -16643.033,E2 -16643.033} C_VEL
LIN {X 0,Y 289.432,Z 549.174,A -85,B 0,C 180,E1 -16645.825,E2 -16645.825} C_VEL
LIN {X 0,Y 289.473,Z 549.678,A -85,B 0,C 180,E1 -16647.219,E2 -16647.219} C_VEL
LIN {X 0,Y 289.496,Z 549.476,A -85,B 0,C 180,E1 -16650.002,E2 -16650.002} C_VEL
LIN {X 0,Y 289.47,Z 548.79,A -85,B 0,C 180,E1 -16651.393,E2 -16651.393} C_VEL
LIN {X 0,Y 289.498,Z 547.684,A -85,B 0,C 180,E1 -16652.785,E2 -16652.785} C_VEL
LIN {X 0,Y 289.487,Z 546.126,A -85,B 0,C 180,E1 -16654.179,E2 -16654.179} C_VEL
LIN {X 0,Y 289.603,Z 542.984,A -85,B 0,C 180,E1 -16656.271,E2 -16656.271} C_VEL
LIN {X 0,Y 289.831,Z 538.751,A -85,B 0,C 180,E1 -16658.368,E2 -16658.368} C_VEL
LIN {X 0,Y 290.388,Z 532.292,A -85,B 0,C 180,E1 -16660.813,E2 -16660.813} C_VEL
LIN {X 0,Y 291.2,Z 525.227,A -85,B 0,C 180,E1 -16662.902,E2 -16662.902} C_VEL
LIN {X 0,Y 292.353,Z 516.356,A -85,B 0,C 180,E1 -16664.978,E2 -16664.978} C_VEL
LIN {X 0,Y 293.616,Z 506.257,A -85,B 0,C 180,E1 -16666.873,E2 -16666.873} C_VEL
LIN {X 0,Y 294.821,Z 495.911,A -85,B 0,C 180,E1 -16668.414,E2 -16668.414} C_VEL
LIN {X 0,Y 296.269,Z 484.452,A -85,B 0,C 180,E1 -16669.759,E2 -16669.759} C_VEL
LIN {X 0,Y 297.518,Z 472.515,A -85,B 0,C 180,E1 -16670.845,E2 -16670.845} C_VEL
LIN {X 0,Y 298.546,Z 460.055,A -85,B 0,C 180,E1 -16671.674,E2 -16671.674} C_VEL
LIN {X 0,Y 299.352,Z 446.336,A -85,B 0,C 180,E1 -16672.286,E2 -16672.286} C_VEL
LIN {X 0,Y 300.717,Z 389.271,A -85,B 0,C 180,E1 -16673.671,E2 -16673.671} C_VEL
LIN {X 0,Y 300.705,Z 379.622,A -85,B 0,C 180,E1 -16673.914,E2 -16673.914} C_VEL
LIN {X 0,Y 295.036,Z 337.108,A -85,B 0,C 180,E1 -16675.392,E2 -16675.392} C_VEL
LIN {X 0,Y 295.334,Z 334.441,A -85,B 0,C 180,E1 -16676.121,E2 -16676.121} C_VEL
LIN {X 0,Y 293.689,Z 324.771,A -85,B 0,C 180,E1 -16678.987,E2 -16678.987} C_VEL
LIN {X 0,Y 291.357,Z 314.187,A -85,B 0,C 180,E1 -16682.282,E2 -16682.282} C_VEL
LIN {X 0,Y 291.368,Z 314.19,A -85,B 0,C 180,E1 -16685.375,E2 -16685.375} C_VEL
LIN {X 0,Y 291.36,Z 314.192,A -85,B 0,C 180,E1 -16688.843,E2 -16688.843} C_VEL
LIN {X 0,Y 291.327,Z 314.198,A -85,B 0,C 180,E1 -16692.493,E2 -16692.493} C_VEL
LIN {X 0,Y 291.316,Z 314.198,A -85,B 0,C 180,E1 -16696.367,E2 -16696.367} C_VEL
LIN {X 0,Y 291.386,Z 314.187,A -85,B 0,C 180,E1 -16700.52,E2 -16700.52} C_VEL
LIN {X 0,Y 291.411,Z 314.186,A -85,B 0,C 180,E1 -16702.92,E2 -16702.92} C_VEL
LIN {X 0,Y 291.352,Z 314.188,A -85,B 0,C 180,E1 -16706.302,E2 -16706.302} C_VEL
LIN {X 0,Y 291.395,Z 314.182,A -85,B 0,C 180,E1 -16710.261,E2 -16710.261} C_VEL
LIN {X 0,Y 291.427,Z 314.181,A -85,B 0,C 180,E1 -16714.273,E2 -16714.273} C_VEL
LIN {X 0,Y 291.379,Z 314.192,A -85,B 0,C 180,E1 -16717.299,E2 -16717.299} C_VEL
LIN {X 0,Y 291.413,Z 314.178,A -85,B 0,C 180,E1 -16720.267,E2 -16720.267} C_VEL
LIN {X 0,Y 291.505,Z 314.168,A -85,B 0,C 180,E1 -16724.665,E2 -16724.665} C_VEL
LIN {X 0,Y 291.542,Z 314.165,A -85,B 0,C 180,E1 -16728.881,E2 -16728.881} C_VEL
LIN {X 0,Y 291.659,Z 314.15,A -85,B 0,C 180,E1 -16731.687,E2 -16731.687} C_VEL
LIN {X 0,Y 291.614,Z 314.152,A -85,B 0,C 180,E1 -16734.468,E2 -16734.468} C_VEL
LIN {X 0,Y 291.894,Z 314.123,A -85,B 0,C 180,E1 -16738.62,E2 -16738.62} C_VEL
LIN {X 0,Y 291.893,Z 314.121,A -85,B 0,C 180,E1 -16741.379,E2 -16741.379} C_VEL
LIN {X 0,Y 291.729,Z 314.136,A -85,B 0,C 180,E1 -16746.918,E2 -16746.918} C_VEL
LIN {X 0,Y 291.575,Z 314.16,A -85,B 0,C 180,E1 -16749.713,E2 -16749.713} C_VEL
LIN {X 0,Y 291.522,Z 314.169,A -85,B 0,C 180,E1 -16753.95,E2 -16753.95} C_VEL
LIN {X 0,Y 291.435,Z 314.183,A -85,B 0,C 180,E1 -16756.821,E2 -16756.821} C_VEL
LIN {X 0,Y 291.43,Z 314.18,A -85,B 0,C 180,E1 -16759.859,E2 -16759.859} C_VEL
LIN {X 0,Y 291.388,Z 314.185,A -85,B 0,C 180,E1 -16764.206,E2 -16764.206} C_VEL
LIN {X 0,Y 291.425,Z 314.182,A -85,B 0,C 180,E1 -16767.271,E2 -16767.271} C_VEL
LIN {X 0,Y 291.34,Z 314.19,A -85,B 0,C 180,E1 -16770.436,E2 -16770.436} C_VEL
LIN {X 0,Y 291.35,Z 314.189,A -85,B 0,C 180,E1 -16773.697,E2 -16773.697} C_VEL
LIN {X 0,Y 291.378,Z 314.19,A -85,B 0,C 180,E1 -16777.252,E2 -16777.252} C_VEL
LIN {X 0,Y 291.354,Z 314.186,A -85,B 0,C 180,E1 -16780.639,E2 -16780.639} C_VEL
LIN {X 0,Y 291.295,Z 314.195,A -85,B 0,C 180,E1 -16784.401,E2 -16784.401} C_VEL
LIN {X 0,Y 291.331,Z 314.192,A -85,B 0,C 180,E1 -16788.403,E2 -16788.403} C_VEL
LIN {X 0,Y 291.368,Z 314.187,A -85,B 0,C 180,E1 -16791.159,E2 -16791.159} C_VEL
LIN {X 0,Y 291.365,Z 314.187,A -85,B 0,C 180,E1 -16794.625,E2 -16794.625} C_VEL
LIN {X 0,Y 291.375,Z 314.191,A -85,B 0,C 180,E1 -16797.949,E2 -16797.949} C_VEL
LIN {X 0,Y 291.381,Z 314.186,A -85,B 0,C 180,E1 -16801.156,E2 -16801.156} C_VEL
LIN {X 0,Y 291.418,Z 314.186,A -85,B 0,C 180,E1 -16804.27,E2 -16804.27} C_VEL
LIN {X 0,Y 291.393,Z 314.185,A -85,B 0,C 180,E1 -16807.299,E2 -16807.299} C_VEL
LIN {X 0,Y 291.466,Z 314.178,A -85,B 0,C 180,E1 -16810.269,E2 -16810.269} C_VEL
LIN {X 0,Y 291.557,Z 314.168,A -85,B 0,C 180,E1 -16814.622,E2 -16814.622} C_VEL
LIN {X 0,Y 291.577,Z 314.275,A -85,B 0,C 180,E1 -16818.528,E2 -16818.528} C_VEL
LIN {X 0,Y 292.146,Z 317.145,A -85,B 0,C 180,E1 -16819.47,E2 -16819.47} C_VEL
LIN {X 0,Y 299.191,Z 337.051,A -85,B 0,C 180,E1 -16820.508,E2 -16820.508} C_VEL
LIN {X 0,Y 301.266,Z 346.587,A -85,B 0,C 180,E1 -16820.893,E2 -16820.893} C_VEL
LIN {X 0,Y 301.433,Z 352.149,A -85,B 0,C 180,E1 -16821.044,E2 -16821.044} C_VEL
LIN {X 0,Y 299.554,Z 425.139,A -85,B 0,C 180,E1 -16822.796,E2 -16822.796} C_VEL
LIN {X 0,Y 298.838,Z 438.881,A -85,B 0,C 180,E1 -16823.415,E2 -16823.415} C_VEL
LIN {X 0,Y 298.057,Z 451.188,A -85,B 0,C 180,E1 -16824.247,E2 -16824.247} C_VEL
LIN {X 0,Y 296.924,Z 463.832,A -85,B 0,C 180,E1 -16825.416,E2 -16825.416} C_VEL
LIN {X 0,Y 295.626,Z 475.641,A -85,B 0,C 180,E1 -16826.834,E2 -16826.834} C_VEL
LIN {X 0,Y 294.381,Z 485.246,A -85,B 0,C 180,E1 -16828.288,E2 -16828.288} C_VEL
LIN {X 0,Y 293.166,Z 494.39,A -85,B 0,C 180,E1 -16829.998,E2 -16829.998} C_VEL
LIN {X 0,Y 291.941,Z 503.308,A -85,B 0,C 180,E1 -16832.067,E2 -16832.067} C_VEL
LIN {X 0,Y 291.053,Z 510.452,A -85,B 0,C 180,E1 -16834.152,E2 -16834.152} C_VEL
LIN {X 0,Y 290.482,Z 516.134,A -85,B 0,C 180,E1 -16836.248,E2 -16836.248} C_VEL
LIN {X 0,Y 289.957,Z 520.627,A -85,B 0,C 180,E1 -16838.36,E2 -16838.36} C_VEL
LIN {X 0,Y 289.676,Z 523.007,A -85,B 0,C 180,E1 -16839.776,E2 -16839.776} C_VEL
LIN {X 0,Y 289.453,Z 524.954,A -85,B 0,C 180,E1 -16841.198,E2 -16841.198} C_VEL
LIN {X 0,Y 289.339,Z 527.252,A -85,B 0,C 180,E1 -16843.69,E2 -16843.69} C_VEL
LIN {X 0,Y 289.262,Z 528.114,A -85,B 0,C 180,E1 -16845.499,E2 -16845.499} C_VEL
LIN {X 0,Y 289.333,Z 528.343,A -85,B 0,C 180,E1 -16846.944,E2 -16846.944} C_VEL
LIN {X 0,Y 289.554,Z 527.978,A -85,B 0,C 180,E1 -16848.809,E2 -16848.809} C_VEL
LIN {X 0,Y 290.032,Z 526.424,A -85,B 0,C 180,E1 -16851.311,E2 -16851.311} C_VEL
LIN {X 0,Y 290.645,Z 524.293,A -85,B 0,C 180,E1 -16853.24,E2 -16853.24} C_VEL
LIN {X 0,Y 291.682,Z 520.405,A -85,B 0,C 180,E1 -16855.7,E2 -16855.7} C_VEL
LIN {X 0,Y 292.928,Z 515.626,A -85,B 0,C 180,E1 -16857.891,E2 -16857.891} C_VEL
LIN {X 0,Y 294.499,Z 509.454,A -85,B 0,C 180,E1 -16860.073,E2 -16860.073} C_VEL
LIN {X 0,Y 296.431,Z 501.668,A -85,B 0,C 180,E1 -16862.236,E2 -16862.236} C_VEL
LIN {X 0,Y 298.348,Z 493.629,A -85,B 0,C 180,E1 -16864.016,E2 -16864.016} C_VEL
LIN {X 0,Y 300.44,Z 483.645,A -85,B 0,C 180,E1 -16865.786,E2 -16865.786} C_VEL
LIN {X 0,Y 302.358,Z 473.803,A -85,B 0,C 180,E1 -16867.178,E2 -16867.178} C_VEL
LIN {X 0,Y 304.239,Z 462.479,A -85,B 0,C 180,E1 -16868.456,E2 -16868.456} C_VEL
LIN {X 0,Y 305.842,Z 450.265,A -85,B 0,C 180,E1 -16869.509,E2 -16869.509} C_VEL
LIN {X 0,Y 307.084,Z 438.115,A -85,B 0,C 180,E1 -16870.274,E2 -16870.274} C_VEL
LIN {X 0,Y 307.979,Z 425.219,A -85,B 0,C 180,E1 -16870.825,E2 -16870.825} C_VEL
LIN {X 0,Y 310.401,Z 354.65,A -85,B 0,C 180,E1 -16872.501,E2 -16872.501} C_VEL
LIN {X 0,Y 303.607,Z 339.31,A -85,B 0,C 180,E1 -16873.759,E2 -16873.759} C_VEL
LIN {X 0,Y 296.644,Z 325.884,A -85,B 0,C 180,E1 -16875.065,E2 -16875.065} C_VEL
LIN {X 0,Y 292.329,Z 318.05,A -85,B 0,C 180,E1 -16875.906,E2 -16875.906} C_VEL
LIN {X 0,Y 291.276,Z 314.2,A -85,B 0,C 180,E1 -16877.5,E2 -16877.5} C_VEL
LIN {X 0,Y 291.321,Z 314.197,A -85,B 0,C 180,E1 -16881.154,E2 -16881.154} C_VEL
LIN {X 0,Y 291.342,Z 314.173,A -85,B 0,C 180,E1 -16884.624,E2 -16884.624} C_VEL
LIN {X 0,Y 291.316,Z 314.192,A -85,B 0,C 180,E1 -16888.416,E2 -16888.416} C_VEL
LIN {X 0,Y 290.606,Z 314.286,A -85,B 0,C 180,E1 -16889.571,E2 -16889.571} C_VEL
LIN {X 0,Y 287.742,Z 314.638,A -85,B 0,C 180,E1 -16891.451,E2 -16891.451} C_VEL
LIN {X 0,Y 285.35,Z 314.939,A -85,B 0,C 180,E1 -16892.978,E2 -16892.978} C_VEL
LIN {X 0,Y 284.341,Z 315.063,A -85,B 0,C 180,E1 -16894.16,E2 -16894.16} C_VEL
LIN {X 0,Y 284.268,Z 315.068,A -85,B 0,C 180,E1 -16894.561,E2 -16894.561} C_VEL
LIN {X 0,Y 284.305,Z 315.064,A -85,B 0,C 180,E1 -16898.235,E2 -16898.235} C_VEL
LIN {X 0,Y 284.39,Z 315.06,A -85,B 0,C 180,E1 -16901.261,E2 -16901.261} C_VEL
LIN {X 0,Y 284.479,Z 315.043,A -85,B 0,C 180,E1 -16904.459,E2 -16904.459} C_VEL
LIN {X 0,Y 284.474,Z 315.039,A -85,B 0,C 180,E1 -16908.601,E2 -16908.601} C_VEL
LIN {X 0,Y 284.598,Z 315.032,A -85,B 0,C 180,E1 -16911.48,E2 -16911.48} C_VEL
LIN {X 0,Y 284.566,Z 315.03,A -85,B 0,C 180,E1 -16914.331,E2 -16914.331} C_VEL
LIN {X 0,Y 284.842,Z 314.99,A -85,B 0,C 180,E1 -16918.586,E2 -16918.586} C_VEL
LIN {X 0,Y 284.843,Z 315,A -85,B 0,C 180,E1 -16921.414,E2 -16921.414} C_VEL
LIN {X 0,Y 284.685,Z 315.016,A -85,B 0,C 180,E1 -16927.091,E2 -16927.091} C_VEL
LIN {X 0,Y 284.554,Z 315.033,A -85,B 0,C 180,E1 -16929.956,E2 -16929.956} C_VEL
LIN {X 0,Y 284.469,Z 315.035,A -85,B 0,C 180,E1 -16934.304,E2 -16934.304} C_VEL
LIN {X 0,Y 284.413,Z 315.053,A -85,B 0,C 180,E1 -16937.249,E2 -16937.249} C_VEL
LIN {X 0,Y 284.367,Z 315.059,A -85,B 0,C 180,E1 -16940.243,E2 -16940.243} C_VEL
LIN {X 0,Y 284.358,Z 315.052,A -85,B 0,C 180,E1 -16943.877,E2 -16943.877} C_VEL
LIN {X 0,Y 284.389,Z 315.053,A -85,B 0,C 180,E1 -16947.176,E2 -16947.176} C_VEL
LIN {X 0,Y 284.288,Z 315.068,A -85,B 0,C 180,E1 -16951.276,E2 -16951.276} C_VEL
LIN {X 0,Y 284.353,Z 315.061,A -85,B 0,C 180,E1 -16955.356,E2 -16955.356} C_VEL
LIN {X 0,Y 284.325,Z 315.07,A -85,B 0,C 180,E1 -16958.167,E2 -16958.167} C_VEL
LIN {X 0,Y 284.296,Z 315.069,A -85,B 0,C 180,E1 -16961.872,E2 -16961.872} C_VEL
LIN {X 0,Y 284.3,Z 315.053,A -85,B 0,C 180,E1 -16965.799,E2 -16965.799} C_VEL
LIN {X 0,Y 284.339,Z 315.069,A -85,B 0,C 180,E1 -16968.14,E2 -16968.14} C_VEL
LIN {X 0,Y 284.367,Z 315.155,A -85,B 0,C 180,E1 -16971.028,E2 -16971.028} C_VEL
LIN {X 0,Y 286.702,Z 323.691,A -85,B 0,C 180,E1 -16974.424,E2 -16974.424} C_VEL
LIN {X 0,Y 288.841,Z 332.374,A -85,B 0,C 180,E1 -16977.639,E2 -16977.639} C_VEL
LIN {X 0,Y 289.558,Z 335.705,A -85,B 0,C 180,E1 -16978.771,E2 -16978.771} C_VEL
LIN {X 0,Y 297.418,Z 352.4,A -85,B 0,C 180,E1 -16980.351,E2 -16980.351} C_VEL
LIN {X 0,Y 299.19,Z 359.92,A -85,B 0,C 180,E1 -16980.8,E2 -16980.8} C_VEL
LIN {X 0,Y 302.772,Z 379.808,A -85,B 0,C 180,E1 -16981.814,E2 -16981.814} C_VEL
LIN {X 0,Y 303.459,Z 385.078,A -85,B 0,C 180,E1 -16982.045,E2 -16982.045} C_VEL
LIN {X 0,Y 301.365,Z 445.213,A -85,B 0,C 180,E1 -16983.515,E2 -16983.515} C_VEL
LIN {X 0,Y 300.182,Z 458.903,A -85,B 0,C 180,E1 -16984.103,E2 -16984.103} C_VEL
LIN {X 0,Y 298.522,Z 471.78,A -85,B 0,C 180,E1 -16984.93,E2 -16984.93} C_VEL
LIN {X 0,Y 296.494,Z 484.28,A -85,B 0,C 180,E1 -16986.053,E2 -16986.053} C_VEL
LIN {X 0,Y 294.38,Z 495.443,A -85,B 0,C 180,E1 -16987.361,E2 -16987.361} C_VEL
LIN {X 0,Y 292.188,Z 505.538,A -85,B 0,C 180,E1 -16988.853,E2 -16988.853} C_VEL
LIN {X 0,Y 289.955,Z 514.664,A -85,B 0,C 180,E1 -16990.535,E2 -16990.535} C_VEL
LIN {X 0,Y 288.326,Z 521.639,A -85,B 0,C 180,E1 -16992.106,E2 -16992.106} C_VEL
LIN {X 0,Y 286.8,Z 528.535,A -85,B 0,C 180,E1 -16994,E2 -16994} C_VEL
LIN {X 0,Y 284.849,Z 535.655,A -85,B 0,C 180,E1 -16996.447,E2 -16996.447} C_VEL
LIN {X 0,Y 283.755,Z 540.426,A -85,B 0,C 180,E1 -16998.574,E2 -16998.574} C_VEL
LIN {X 0,Y 283.032,Z 544.105,A -85,B 0,C 180,E1 -17000.714,E2 -17000.714} C_VEL
LIN {X 0,Y 282.556,Z 546.793,A -85,B 0,C 180,E1 -17002.858,E2 -17002.858} C_VEL
LIN {X 0,Y 282.402,Z 548.276,A -85,B 0,C 180,E1 -17004.542,E2 -17004.542} C_VEL
LIN {X 0,Y 282.377,Z 549.425,A -85,B 0,C 180,E1 -17007.149,E2 -17007.149} C_VEL
LIN {X 0,Y 282.367,Z 549.491,A -85,B 0,C 180,E1 -17008.576,E2 -17008.576} C_VEL
LIN {X 0,Y 282.413,Z 549.173,A -85,B 0,C 180,E1 -17010.002,E2 -17010.002} C_VEL
LIN {X 0,Y 282.391,Z 548.46,A -85,B 0,C 180,E1 -17011.428,E2 -17011.428} C_VEL
LIN {X 0,Y 282.425,Z 547.305,A -85,B 0,C 180,E1 -17012.855,E2 -17012.855} C_VEL
LIN {X 0,Y 282.44,Z 543.976,A -85,B 0,C 180,E1 -17015.538,E2 -17015.538} C_VEL
LIN {X 0,Y 282.669,Z 539.794,A -85,B 0,C 180,E1 -17017.862,E2 -17017.862} C_VEL
LIN {X 0,Y 283.08,Z 534.718,A -85,B 0,C 180,E1 -17020.01,E2 -17020.01} C_VEL
LIN {X 0,Y 283.717,Z 528.314,A -85,B 0,C 180,E1 -17022.157,E2 -17022.157} C_VEL
LIN {X 0,Y 284.798,Z 520.282,A -85,B 0,C 180,E1 -17024.289,E2 -17024.289} C_VEL
LIN {X 0,Y 286.042,Z 511.118,A -85,B 0,C 180,E1 -17026.243,E2 -17026.243} C_VEL
LIN {X 0,Y 287.37,Z 500.931,A -85,B 0,C 180,E1 -17027.987,E2 -17027.987} C_VEL
LIN {X 0,Y 288.628,Z 490.748,A -85,B 0,C 180,E1 -17029.378,E2 -17029.378} C_VEL
LIN {X 0,Y 289.896,Z 479.649,A -85,B 0,C 180,E1 -17030.583,E2 -17030.583} C_VEL
LIN {X 0,Y 291.17,Z 467.368,A -85,B 0,C 180,E1 -17031.6,E2 -17031.6} C_VEL
LIN {X 0,Y 292.156,Z 454.471,A -85,B 0,C 180,E1 -17032.359,E2 -17032.359} C_VEL
LIN {X 0,Y 292.803,Z 440.575,A -85,B 0,C 180,E1 -17032.872,E2 -17032.872} C_VEL
LIN {X 0,Y 294.168,Z 381.843,A -85,B 0,C 180,E1 -17034.295,E2 -17034.295} C_VEL
LIN {X 0,Y 288.248,Z 336.82,A -85,B 0,C 180,E1 -17035.908,E2 -17035.908} C_VEL
LIN {X 0,Y 288.124,Z 333.665,A -85,B 0,C 180,E1 -17036.826,E2 -17036.826} C_VEL
LIN {X 0,Y 286.137,Z 323.462,A -85,B 0,C 180,E1 -17039.97,E2 -17039.97} C_VEL
LIN {X 0,Y 284.297,Z 315.065,A -85,B 0,C 180,E1 -17042.68,E2 -17042.68} C_VEL
LIN {X 0,Y 284.339,Z 315.067,A -85,B 0,C 180,E1 -17046.387,E2 -17046.387} C_VEL
LIN {X 0,Y 284.313,Z 315.07,A -85,B 0,C 180,E1 -17049.996,E2 -17049.996} C_VEL
LIN {X 0,Y 284.253,Z 315.077,A -85,B 0,C 180,E1 -17054.191,E2 -17054.191} C_VEL
LIN {X 0,Y 284.279,Z 315.072,A -85,B 0,C 180,E1 -17058.125,E2 -17058.125} C_VEL
LIN {X 0,Y 284.326,Z 315.065,A -85,B 0,C 180,E1 -17062.28,E2 -17062.28} C_VEL
LIN {X 0,Y 284.316,Z 315.066,A -85,B 0,C 180,E1 -17065.351,E2 -17065.351} C_VEL
LIN {X 0,Y 284.303,Z 315.07,A -85,B 0,C 180,E1 -17068.726,E2 -17068.726} C_VEL
LIN {X 0,Y 284.407,Z 315.057,A -85,B 0,C 180,E1 -17072.826,E2 -17072.826} C_VEL
LIN {X 0,Y 284.34,Z 315.064,A -85,B 0,C 180,E1 -17076.704,E2 -17076.704} C_VEL
LIN {X 0,Y 284.384,Z 315.054,A -85,B 0,C 180,E1 -17079.905,E2 -17079.905} C_VEL
LIN {X 0,Y 284.454,Z 315.047,A -85,B 0,C 180,E1 -17084.493,E2 -17084.493} C_VEL
LIN {X 0,Y 284.494,Z 315.043,A -85,B 0,C 180,E1 -17088.601,E2 -17088.601} C_VEL
LIN {X 0,Y 284.616,Z 315.027,A -85,B 0,C 180,E1 -17091.48,E2 -17091.48} C_VEL
LIN {X 0,Y 284.583,Z 315.028,A -85,B 0,C 180,E1 -17094.331,E2 -17094.331} C_VEL
LIN {X 0,Y 284.86,Z 314.999,A -85,B 0,C 180,E1 -17098.586,E2 -17098.586} C_VEL
LIN {X 0,Y 284.86,Z 314.997,A -85,B 0,C 180,E1 -17101.413,E2 -17101.413} C_VEL
LIN {X 0,Y 284.68,Z 315.013,A -85,B 0,C 180,E1 -17107.09,E2 -17107.09} C_VEL
LIN {X 0,Y 284.521,Z 315.039,A -85,B 0,C 180,E1 -17109.957,E2 -17109.957} C_VEL
LIN {X 0,Y 284.47,Z 315.05,A -85,B 0,C 180,E1 -17114.303,E2 -17114.303} C_VEL
LIN {X 0,Y 284.347,Z 315.068,A -85,B 0,C 180,E1 -17118.742,E2 -17118.742} C_VEL
LIN {X 0,Y 284.319,Z 315.064,A -85,B 0,C 180,E1 -17121.763,E2 -17121.763} C_VEL
LIN {X 0,Y 284.342,Z 315.067,A -85,B 0,C 180,E1 -17124.846,E2 -17124.846} C_VEL
LIN {X 0,Y 284.333,Z 315.062,A -85,B 0,C 180,E1 -17128.01,E2 -17128.01} C_VEL
LIN {X 0,Y 284.3,Z 315.072,A -85,B 0,C 180,E1 -17131.273,E2 -17131.273} C_VEL
LIN {X 0,Y 284.346,Z 315.064,A -85,B 0,C 180,E1 -17135.347,E2 -17135.347} C_VEL
LIN {X 0,Y 284.314,Z 315.065,A -85,B 0,C 180,E1 -17138.168,E2 -17138.168} C_VEL
LIN {X 0,Y 284.288,Z 315.069,A -85,B 0,C 180,E1 -17142.126,E2 -17142.126} C_VEL
LIN {X 0,Y 284.26,Z 315.073,A -85,B 0,C 180,E1 -17146.188,E2 -17146.188} C_VEL
LIN {X 0,Y 284.312,Z 315.068,A -85,B 0,C 180,E1 -17150.022,E2 -17150.022} C_VEL
LIN {X 0,Y 284.339,Z 315.067,A -85,B 0,C 180,E1 -17153.613,E2 -17153.613} C_VEL
LIN {X 0,Y 284.311,Z 315.067,A -85,B 0,C 180,E1 -17157.188,E2 -17157.188} C_VEL
LIN {X 0,Y 284.359,Z 315.064,A -85,B 0,C 180,E1 -17160.374,E2 -17160.374} C_VEL
LIN {X 0,Y 284.38,Z 315.06,A -85,B 0,C 180,E1 -17163.585,E2 -17163.585} C_VEL
LIN {X 0,Y 284.373,Z 315.062,A -85,B 0,C 180,E1 -17166.706,E2 -17166.706} C_VEL
LIN {X 0,Y 284.409,Z 315.056,A -85,B 0,C 180,E1 -17171.26,E2 -17171.26} C_VEL
LIN {X 0,Y 284.495,Z 315.048,A -85,B 0,C 180,E1 -17174.457,E2 -17174.457} C_VEL
LIN {X 0,Y 284.498,Z 315.126,A -85,B 0,C 180,E1 -17178.148,E2 -17178.148} C_VEL
LIN {X 0,Y 285.003,Z 317.486,A -85,B 0,C 180,E1 -17178.934,E2 -17178.934} C_VEL
LIN {X 0,Y 292.751,Z 339.182,A -85,B 0,C 180,E1 -17180.1,E2 -17180.1} C_VEL
LIN {X 0,Y 294.516,Z 347.136,A -85,B 0,C 180,E1 -17180.434,E2 -17180.434} C_VEL
LIN {X 0,Y 294.815,Z 350.549,A -85,B 0,C 180,E1 -17180.544,E2 -17180.544} C_VEL
LIN {X 0,Y 292.807,Z 425.205,A -85,B 0,C 180,E1 -17182.369,E2 -17182.369} C_VEL
LIN {X 0,Y 292.067,Z 439.01,A -85,B 0,C 180,E1 -17183.001,E2 -17183.001} C_VEL
LIN {X 0,Y 291.258,Z 451.356,A -85,B 0,C 180,E1 -17183.851,E2 -17183.851} C_VEL
LIN {X 0,Y 290.158,Z 463.235,A -85,B 0,C 180,E1 -17184.961,E2 -17184.961} C_VEL
LIN {X 0,Y 288.911,Z 474.668,A -85,B 0,C 180,E1 -17186.34,E2 -17186.34} C_VEL
LIN {X 0,Y 287.565,Z 484.954,A -85,B 0,C 180,E1 -17187.897,E2 -17187.897} C_VEL
LIN {X 0,Y 286.281,Z 494.202,A -85,B 0,C 180,E1 -17189.646,E2 -17189.646} C_VEL
LIN {X 0,Y 284.981,Z 503.199,A -85,B 0,C 180,E1 -17191.764,E2 -17191.764} C_VEL
LIN {X 0,Y 284.042,Z 510.428,A -85,B 0,C 180,E1 -17193.899,E2 -17193.899} C_VEL
LIN {X 0,Y 283.375,Z 516.788,A -85,B 0,C 180,E1 -17196.317,E2 -17196.317} C_VEL
LIN {X 0,Y 282.833,Z 521.351,A -85,B 0,C 180,E1 -17198.572,E2 -17198.572} C_VEL
LIN {X 0,Y 282.543,Z 523.67,A -85,B 0,C 180,E1 -17200.025,E2 -17200.025} C_VEL
LIN {X 0,Y 282.351,Z 525.516,A -85,B 0,C 180,E1 -17201.484,E2 -17201.484} C_VEL
LIN {X 0,Y 282.241,Z 527.536,A -85,B 0,C 180,E1 -17203.803,E2 -17203.803} C_VEL
LIN {X 0,Y 282.17,Z 528.469,A -85,B 0,C 180,E1 -17205.899,E2 -17205.899} C_VEL
LIN {X 0,Y 282.28,Z 528.586,A -85,B 0,C 180,E1 -17207.381,E2 -17207.381} C_VEL
LIN {X 0,Y 282.486,Z 528.247,A -85,B 0,C 180,E1 -17209.021,E2 -17209.021} C_VEL
LIN {X 0,Y 282.714,Z 527.597,A -85,B 0,C 180,E1 -17210.364,E2 -17210.364} C_VEL
LIN {X 0,Y 283.086,Z 526.435,A -85,B 0,C 180,E1 -17211.861,E2 -17211.861} C_VEL
LIN {X 0,Y 283.669,Z 524.571,A -85,B 0,C 180,E1 -17213.554,E2 -17213.554} C_VEL
LIN {X 0,Y 284.546,Z 521.494,A -85,B 0,C 180,E1 -17215.607,E2 -17215.607} C_VEL
LIN {X 0,Y 285.807,Z 516.993,A -85,B 0,C 180,E1 -17217.851,E2 -17217.851} C_VEL
LIN {X 0,Y 287.398,Z 511.168,A -85,B 0,C 180,E1 -17220.084,E2 -17220.084} C_VEL
LIN {X 0,Y 289.378,Z 503.737,A -85,B 0,C 180,E1 -17222.294,E2 -17222.294} C_VEL
LIN {X 0,Y 291.302,Z 496.068,A -85,B 0,C 180,E1 -17224.117,E2 -17224.117} C_VEL
LIN {X 0,Y 293.589,Z 485.949,A -85,B 0,C 180,E1 -17226.053,E2 -17226.053} C_VEL
LIN {X 0,Y 295.677,Z 476.199,A -85,B 0,C 180,E1 -17227.52,E2 -17227.52} C_VEL
LIN {X 0,Y 297.565,Z 465.638,A -85,B 0,C 180,E1 -17228.794,E2 -17228.794} C_VEL
LIN {X 0,Y 299.375,Z 452.953,A -85,B 0,C 180,E1 -17229.986,E2 -17229.986} C_VEL
LIN {X 0,Y 300.654,Z 441.707,A -85,B 0,C 180,E1 -17230.769,E2 -17230.769} C_VEL
LIN {X 0,Y 301.72,Z 428.721,A -85,B 0,C 180,E1 -17231.392,E2 -17231.392} C_VEL
LIN {X 0,Y 302.522,Z 411.763,A -85,B 0,C 180,E1 -17231.857,E2 -17231.857} C_VEL
LIN {X 0,Y 304.427,Z 356.712,A -85,B 0,C 180,E1 -17233.166,E2 -17233.166} C_VEL
LIN {X 0,Y 297.77,Z 341.916,A -85,B 0,C 180,E1 -17234.442,E2 -17234.442} C_VEL
LIN {X 0,Y 291.427,Z 329.682,A -85,B 0,C 180,E1 -17235.679,E2 -17235.679} C_VEL
LIN {X 0,Y 285.137,Z 318.331,A -85,B 0,C 180,E1 -17236.985,E2 -17236.985} C_VEL
LIN {X 0,Y 284.253,Z 315.078,A -85,B 0,C 180,E1 -17238.359,E2 -17238.359} C_VEL
LIN {X 0,Y 284.292,Z 315.076,A -85,B 0,C 180,E1 -17242.281,E2 -17242.281} C_VEL
LIN {X 0,Y 284.294,Z 315.054,A -85,B 0,C 180,E1 -17245.349,E2 -17245.349} C_VEL
LIN {X 0,Y 284.272,Z 315.069,A -85,B 0,C 180,E1 -17248.723,E2 -17248.723} C_VEL
LIN {X 0,Y 284.27,Z 315.069,A -85,B 0,C 180,E1 -17251.983,E2 -17251.983} C_VEL
LIN {X 0,Y 284.268,Z 315.068,A -85,B 0,C 180,E1 -17254.561,E2 -17254.561} C_VEL
LIN {X 0,Y 283.638,Z 315.147,A -85,B 0,C 180,E1 -17255.742,E2 -17255.742} C_VEL
LIN {X 0,Y 280.86,Z 315.503,A -85,B 0,C 180,E1 -17257.669,E2 -17257.669} C_VEL
LIN {X 0,Y 278.473,Z 315.805,A -85,B 0,C 180,E1 -17259.234,E2 -17259.234} C_VEL
LIN {X 0,Y 277.425,Z 315.931,A -85,B 0,C 180,E1 -17260.445,E2 -17260.445} C_VEL
LIN {X 0,Y 277.327,Z 315.939,A -85,B 0,C 180,E1 -17260.855,E2 -17260.855} C_VEL
LIN {X 0,Y 277.421,Z 315.927,A -85,B 0,C 180,E1 -17265.325,E2 -17265.325} C_VEL
LIN {X 0,Y 277.447,Z 315.922,A -85,B 0,C 180,E1 -17269.787,E2 -17269.787} C_VEL
LIN {X 0,Y 277.592,Z 315.892,A -85,B 0,C 180,E1 -17272.728,E2 -17272.728} C_VEL
LIN {X 0,Y 277.808,Z 315.866,A -85,B 0,C 180,E1 -17278.551,E2 -17278.551} C_VEL
LIN {X 0,Y 277.809,Z 315.876,A -85,B 0,C 180,E1 -17281.45,E2 -17281.45} C_VEL
LIN {X 0,Y 277.64,Z 315.893,A -85,B 0,C 180,E1 -17287.272,E2 -17287.272} C_VEL
LIN {X 0,Y 277.494,Z 315.913,A -85,B 0,C 180,E1 -17290.212,E2 -17290.212} C_VEL
LIN {X 0,Y 277.422,Z 315.916,A -85,B 0,C 180,E1 -17294.675,E2 -17294.675} C_VEL
LIN {X 0,Y 277.333,Z 315.927,A -85,B 0,C 180,E1 -17299.235,E2 -17299.235} C_VEL
LIN {X 0,Y 277.308,Z 315.931,A -85,B 0,C 180,E1 -17304.172,E2 -17304.172} C_VEL
LIN {X 0,Y 277.317,Z 315.931,A -85,B 0,C 180,E1 -17307.508,E2 -17307.508} C_VEL
LIN {X 0,Y 277.262,Z 315.949,A -85,B 0,C 180,E1 -17310.483,E2 -17310.483} C_VEL
LIN {X 0,Y 277.245,Z 315.953,A -85,B 0,C 180,E1 -17313.896,E2 -17313.896} C_VEL
LIN {X 0,Y 277.281,Z 315.95,A -85,B 0,C 180,E1 -17317.468,E2 -17317.468} C_VEL
LIN {X 0,Y 277.234,Z 315.953,A -85,B 0,C 180,E1 -17321.233,E2 -17321.233} C_VEL
LIN {X 0,Y 277.242,Z 315.934,A -85,B 0,C 180,E1 -17325.218,E2 -17325.218} C_VEL
LIN {X 0,Y 277.29,Z 315.933,A -85,B 0,C 180,E1 -17329.496,E2 -17329.496} C_VEL
LIN {X 0,Y 277.318,Z 315.95,A -85,B 0,C 180,E1 -17330.026,E2 -17330.026} C_VEL
LIN {X 0,Y 279.89,Z 325.322,A -85,B 0,C 180,E1 -17333.906,E2 -17333.906} C_VEL
LIN {X 0,Y 282.293,Z 335.223,A -85,B 0,C 180,E1 -17337.666,E2 -17337.666} C_VEL
LIN {X 0,Y 284.308,Z 339.393,A -85,B 0,C 180,E1 -17338.109,E2 -17338.109} C_VEL
LIN {X 0,Y 291.415,Z 354.382,A -85,B 0,C 180,E1 -17339.599,E2 -17339.599} C_VEL
LIN {X 0,Y 292.578,Z 357.606,A -85,B 0,C 180,E1 -17339.855,E2 -17339.855} C_VEL
LIN {X 0,Y 296.694,Z 380.091,A -85,B 0,C 180,E1 -17341.061,E2 -17341.061} C_VEL
LIN {X 0,Y 297.45,Z 386.688,A -85,B 0,C 180,E1 -17341.348,E2 -17341.348} C_VEL
LIN {X 0,Y 295.343,Z 444.77,A -85,B 0,C 180,E1 -17342.791,E2 -17342.791} C_VEL
LIN {X 0,Y 294.223,Z 457.701,A -85,B 0,C 180,E1 -17343.347,E2 -17343.347} C_VEL
LIN {X 0,Y 292.485,Z 470.867,A -85,B 0,C 180,E1 -17344.184,E2 -17344.184} C_VEL
LIN {X 0,Y 290.663,Z 481.958,A -85,B 0,C 180,E1 -17345.161,E2 -17345.161} C_VEL
LIN {X 0,Y 288.385,Z 493.5,A -85,B 0,C 180,E1 -17346.483,E2 -17346.483} C_VEL
LIN {X 0,Y 286.081,Z 503.908,A -85,B 0,C 180,E1 -17348.001,E2 -17348.001} C_VEL
LIN {X 0,Y 283.753,Z 513.319,A -85,B 0,C 180,E1 -17349.714,E2 -17349.714} C_VEL
LIN {X 0,Y 281.767,Z 520.871,A -85,B 0,C 180,E1 -17351.41,E2 -17351.41} C_VEL
LIN {X 0,Y 279.969,Z 528.639,A -85,B 0,C 180,E1 -17353.599,E2 -17353.599} C_VEL
LIN {X 0,Y 277.938,Z 535.684,A -85,B 0,C 180,E1 -17356.103,E2 -17356.103} C_VEL
LIN {X 0,Y 276.773,Z 540.392,A -85,B 0,C 180,E1 -17358.282,E2 -17358.282} C_VEL
LIN {X 0,Y 275.992,Z 544.013,A -85,B 0,C 180,E1 -17360.475,E2 -17360.475} C_VEL
LIN {X 0,Y 275.493,Z 546.645,A -85,B 0,C 180,E1 -17362.674,E2 -17362.674} C_VEL
LIN {X 0,Y 275.321,Z 548.191,A -85,B 0,C 180,E1 -17364.588,E2 -17364.588} C_VEL
LIN {X 0,Y 275.284,Z 549.172,A -85,B 0,C 180,E1 -17367.075,E2 -17367.075} C_VEL
LIN {X 0,Y 275.29,Z 549.213,A -85,B 0,C 180,E1 -17368.539,E2 -17368.539} C_VEL
LIN {X 0,Y 275.332,Z 548.869,A -85,B 0,C 180,E1 -17370.002,E2 -17370.002} C_VEL
LIN {X 0,Y 275.315,Z 548.117,A -85,B 0,C 180,E1 -17371.465,E2 -17371.465} C_VEL
LIN {X 0,Y 275.352,Z 546.921,A -85,B 0,C 180,E1 -17372.928,E2 -17372.928} C_VEL
LIN {X 0,Y 275.362,Z 543.799,A -85,B 0,C 180,E1 -17375.5,E2 -17375.5} C_VEL
LIN {X 0,Y 275.593,Z 539.291,A -85,B 0,C 180,E1 -17378.065,E2 -17378.065} C_VEL
LIN {X 0,Y 276.139,Z 533.143,A -85,B 0,C 180,E1 -17380.635,E2 -17380.635} C_VEL
LIN {X 0,Y 276.901,Z 526.395,A -85,B 0,C 180,E1 -17382.833,E2 -17382.833} C_VEL
LIN {X 0,Y 278.057,Z 518.012,A -85,B 0,C 180,E1 -17385.017,E2 -17385.017} C_VEL
LIN {X 0,Y 279.226,Z 509.48,A -85,B 0,C 180,E1 -17386.806,E2 -17386.806} C_VEL
LIN {X 0,Y 280.678,Z 498.687,A -85,B 0,C 180,E1 -17388.62,E2 -17388.62} C_VEL
LIN {X 0,Y 281.859,Z 489.527,A -85,B 0,C 180,E1 -17389.863,E2 -17389.863} C_VEL
LIN {X 0,Y 283.191,Z 478.204,A -85,B 0,C 180,E1 -17391.093,E2 -17391.093} C_VEL
LIN {X 0,Y 284.545,Z 465.47,A -85,B 0,C 180,E1 -17392.129,E2 -17392.129} C_VEL
LIN {X 0,Y 285.526,Z 452.711,A -85,B 0,C 180,E1 -17392.86,E2 -17392.86} C_VEL
LIN {X 0,Y 286.104,Z 439.748,A -85,B 0,C 180,E1 -17393.331,E2 -17393.331} C_VEL
LIN {X 0,Y 287.447,Z 382.047,A -85,B 0,C 180,E1 -17394.761,E2 -17394.761} C_VEL
LIN {X 0,Y 281.709,Z 338.543,A -85,B 0,C 180,E1 -17396.358,E2 -17396.358} C_VEL
LIN {X 0,Y 281.342,Z 336.473,A -85,B 0,C 180,E1 -17396.476,E2 -17396.476} C_VEL
LIN {X 0,Y 279.755,Z 327.323,A -85,B 0,C 180,E1 -17399.334,E2 -17399.334} C_VEL
LIN {X 0,Y 277.259,Z 315.942,A -85,B 0,C 180,E1 -17403.1,E2 -17403.1} C_VEL
LIN {X 0,Y 277.287,Z 315.944,A -85,B 0,C 180,E1 -17405.8,E2 -17405.8} C_VEL
LIN {X 0,Y 277.241,Z 315.949,A -85,B 0,C 180,E1 -17409.329,E2 -17409.329} C_VEL
LIN {X 0,Y 277.216,Z 315.952,A -85,B 0,C 180,E1 -17413.199,E2 -17413.199} C_VEL
LIN {X 0,Y 277.222,Z 315.951,A -85,B 0,C 180,E1 -17417.326,E2 -17417.326} C_VEL
LIN {X 0,Y 277.269,Z 315.943,A -85,B 0,C 180,E1 -17421.794,E2 -17421.794} C_VEL
LIN {X 0,Y 277.291,Z 315.941,A -85,B 0,C 180,E1 -17424.342,E2 -17424.342} C_VEL
LIN {X 0,Y 277.252,Z 315.946,A -85,B 0,C 180,E1 -17427.837,E2 -17427.837} C_VEL
LIN {X 0,Y 277.298,Z 315.944,A -85,B 0,C 180,E1 -17431.213,E2 -17431.213} C_VEL
LIN {X 0,Y 277.319,Z 315.938,A -85,B 0,C 180,E1 -17434.48,E2 -17434.48} C_VEL
LIN {X 0,Y 277.272,Z 315.946,A -85,B 0,C 180,E1 -17437.653,E2 -17437.653} C_VEL
LIN {X 0,Y 277.312,Z 315.934,A -85,B 0,C 180,E1 -17440.763,E2 -17440.763} C_VEL
LIN {X 0,Y 277.417,Z 315.926,A -85,B 0,C 180,E1 -17445.325,E2 -17445.325} C_VEL
LIN {X 0,Y 277.468,Z 315.92,A -85,B 0,C 180,E1 -17449.787,E2 -17449.787} C_VEL
LIN {X 0,Y 277.609,Z 315.89,A -85,B 0,C 180,E1 -17452.728,E2 -17452.728} C_VEL
LIN {X 0,Y 277.826,Z 315.875,A -85,B 0,C 180,E1 -17458.55,E2 -17458.55} C_VEL
LIN {X 0,Y 277.826,Z 315.874,A -85,B 0,C 180,E1 -17461.449,E2 -17461.449} C_VEL
LIN {X 0,Y 277.634,Z 315.889,A -85,B 0,C 180,E1 -17467.271,E2 -17467.271} C_VEL
LIN {X 0,Y 277.464,Z 315.92,A -85,B 0,C 180,E1 -17470.213,E2 -17470.213} C_VEL
LIN {X 0,Y 277.416,Z 315.927,A -85,B 0,C 180,E1 -17474.675,E2 -17474.675} C_VEL
LIN {X 0,Y 277.311,Z 315.94,A -85,B 0,C 180,E1 -17479.236,E2 -17479.236} C_VEL
LIN {X 0,Y 277.303,Z 315.939,A -85,B 0,C 180,E1 -17483.923,E2 -17483.923} C_VEL
LIN {X 0,Y 277.329,Z 315.936,A -85,B 0,C 180,E1 -17487.503,E2 -17487.503} C_VEL
LIN {X 0,Y 277.278,Z 315.942,A -85,B 0,C 180,E1 -17490.48,E2 -17490.48} C_VEL
LIN {X 0,Y 277.253,Z 315.943,A -85,B 0,C 180,E1 -17493.895,E2 -17493.895} C_VEL
LIN {X 0,Y 277.271,Z 315.947,A -85,B 0,C 180,E1 -17497.469,E2 -17497.469} C_VEL
LIN {X 0,Y 277.225,Z 315.949,A -85,B 0,C 180,E1 -17501.233,E2 -17501.233} C_VEL
LIN {X 0,Y 277.206,Z 315.952,A -85,B 0,C 180,E1 -17505.225,E2 -17505.225} C_VEL
LIN {X 0,Y 277.228,Z 315.952,A -85,B 0,C 180,E1 -17509.511,E2 -17509.511} C_VEL
LIN {X 0,Y 277.276,Z 315.944,A -85,B 0,C 180,E1 -17512.53,E2 -17512.53} C_VEL
LIN {X 0,Y 277.251,Z 315.951,A -85,B 0,C 180,E1 -17516.103,E2 -17516.103} C_VEL
LIN {X 0,Y 277.265,Z 315.945,A -85,B 0,C 180,E1 -17519.537,E2 -17519.537} C_VEL
LIN {X 0,Y 277.36,Z 315.934,A -85,B 0,C 180,E1 -17522.862,E2 -17522.862} C_VEL
LIN {X 0,Y 277.333,Z 315.94,A -85,B 0,C 180,E1 -17526.078,E2 -17526.078} C_VEL
LIN {X 0,Y 277.35,Z 315.938,A -85,B 0,C 180,E1 -17530.765,E2 -17530.765} C_VEL
LIN {X 0,Y 277.437,Z 315.926,A -85,B 0,C 180,E1 -17535.324,E2 -17535.324} C_VEL
LIN {X 0,Y 277.459,Z 315.974,A -85,B 0,C 180,E1 -17537.75,E2 -17537.75} C_VEL
LIN {X 0,Y 277.825,Z 317.678,A -85,B 0,C 180,E1 -17538.347,E2 -17538.347} C_VEL
LIN {X 0,Y 285.47,Z 338.806,A -85,B 0,C 180,E1 -17539.543,E2 -17539.543} C_VEL
LIN {X 0,Y 287.299,Z 345.058,A -85,B 0,C 180,E1 -17539.848,E2 -17539.848} C_VEL
LIN {X 0,Y 288.144,Z 349.718,A -85,B 0,C 180,E1 -17540.035,E2 -17540.035} C_VEL
LIN {X 0,Y 286.077,Z 425.27,A -85,B 0,C 180,E1 -17541.922,E2 -17541.922} C_VEL
LIN {X 0,Y 285.352,Z 438.386,A -85,B 0,C 180,E1 -17542.524,E2 -17542.524} C_VEL
LIN {X 0,Y 284.49,Z 451.515,A -85,B 0,C 180,E1 -17543.437,E2 -17543.437} C_VEL
LIN {X 0,Y 283.414,Z 462.637,A -85,B 0,C 180,E1 -17544.484,E2 -17544.484} C_VEL
LIN {X 0,Y 282.084,Z 474.669,A -85,B 0,C 180,E1 -17545.956,E2 -17545.956} C_VEL
LIN {X 0,Y 280.728,Z 484.637,A -85,B 0,C 180,E1 -17547.487,E2 -17547.487} C_VEL
LIN {X 0,Y 279.386,Z 494.018,A -85,B 0,C 180,E1 -17549.277,E2 -17549.277} C_VEL
LIN {X 0,Y 278.05,Z 503.086,A -85,B 0,C 180,E1 -17551.446,E2 -17551.446} C_VEL
LIN {X 0,Y 277.054,Z 510.387,A -85,B 0,C 180,E1 -17553.634,E2 -17553.634} C_VEL
LIN {X 0,Y 276.402,Z 516.212,A -85,B 0,C 180,E1 -17555.835,E2 -17555.835} C_VEL
LIN {X 0,Y 275.86,Z 520.808,A -85,B 0,C 180,E1 -17558.053,E2 -17558.053} C_VEL
LIN {X 0,Y 275.411,Z 524.313,A -85,B 0,C 180,E1 -17560.287,E2 -17560.287} C_VEL
LIN {X 0,Y 275.231,Z 526.054,A -85,B 0,C 180,E1 -17561.785,E2 -17561.785} C_VEL
LIN {X 0,Y 275.153,Z 527.822,A -85,B 0,C 180,E1 -17563.928,E2 -17563.928} C_VEL
LIN {X 0,Y 275.114,Z 528.774,A -85,B 0,C 180,E1 -17566.318,E2 -17566.318} C_VEL
LIN {X 0,Y 275.435,Z 528.513,A -85,B 0,C 180,E1 -17569.25,E2 -17569.25} C_VEL
LIN {X 0,Y 275.74,Z 527.687,A -85,B 0,C 180,E1 -17570.903,E2 -17570.903} C_VEL
LIN {X 0,Y 276.191,Z 526.431,A -85,B 0,C 180,E1 -17572.436,E2 -17572.436} C_VEL
LIN {X 0,Y 277.059,Z 523.708,A -85,B 0,C 180,E1 -17574.74,E2 -17574.74} C_VEL
LIN {X 0,Y 278.206,Z 519.867,A -85,B 0,C 180,E1 -17577.044,E2 -17577.044} C_VEL
LIN {X 0,Y 279.695,Z 514.783,A -85,B 0,C 180,E1 -17579.337,E2 -17579.337} C_VEL
LIN {X 0,Y 281.588,Z 508.294,A -85,B 0,C 180,E1 -17581.607,E2 -17581.607} C_VEL
LIN {X 0,Y 283.812,Z 500.02,A -85,B 0,C 180,E1 -17583.857,E2 -17583.857} C_VEL
LIN {X 0,Y 286.174,Z 490.68,A -85,B 0,C 180,E1 -17585.863,E2 -17585.863} C_VEL
LIN {X 0,Y 288.421,Z 480.909,A -85,B 0,C 180,E1 -17587.527,E2 -17587.527} C_VEL
LIN {X 0,Y 290.538,Z 470.254,A -85,B 0,C 180,E1 -17588.968,E2 -17588.968} C_VEL
LIN {X 0,Y 292.589,Z 458.112,A -85,B 0,C 180,E1 -17590.249,E2 -17590.249} C_VEL
LIN {X 0,Y 294.055,Z 446.268,A -85,B 0,C 180,E1 -17591.201,E2 -17591.201} C_VEL
LIN {X 0,Y 295.419,Z 432.598,A -85,B 0,C 180,E1 -17591.955,E2 -17591.955} C_VEL
LIN {X 0,Y 296.177,Z 419.841,A -85,B 0,C 180,E1 -17592.394,E2 -17592.394} C_VEL
LIN {X 0,Y 298.439,Z 358.825,A -85,B 0,C 180,E1 -17593.862,E2 -17593.862} C_VEL
LIN {X 0,Y 292.942,Z 346.384,A -85,B 0,C 180,E1 -17594.964,E2 -17594.964} C_VEL
LIN {X 0,Y 286.666,Z 334.099,A -85,B 0,C 180,E1 -17596.238,E2 -17596.238} C_VEL
LIN {X 0,Y 279.928,Z 322.314,A -85,B 0,C 180,E1 -17597.659,E2 -17597.659} C_VEL
LIN {X 0,Y 277.898,Z 318.59,A -85,B 0,C 180,E1 -17598.163,E2 -17598.163} C_VEL
LIN {X 0,Y 277.226,Z 315.954,A -85,B 0,C 180,E1 -17599.342,E2 -17599.342} C_VEL
LIN {X 0,Y 277.239,Z 315.95,A -85,B 0,C 180,E1 -17602.526,E2 -17602.526} C_VEL
LIN {X 0,Y 277.233,Z 315.942,A -85,B 0,C 180,E1 -17606.103,E2 -17606.103} C_VEL
LIN {X 0,Y 277.25,Z 315.947,A -85,B 0,C 180,E1 -17609.537,E2 -17609.537} C_VEL
LIN {X 0,Y 277.279,Z 315.945,A -85,B 0,C 180,E1 -17612.856,E2 -17612.856} C_VEL
LIN {X 0,Y 277.269,Z 315.942,A -85,B 0,C 180,E1 -17616.074,E2 -17616.074} C_VEL
LIN {X 0,Y 277.332,Z 315.939,A -85,B 0,C 180,E1 -17620.766,E2 -17620.766} C_VEL
LIN {X 0,Y 277.327,Z 315.939,A -85,B 0,C 180,E1 -17620.855,E2 -17620.855} C_VEL
LIN {X 0,Y 276.629,Z 316.023,A -85,B 0,C 180,E1 -17622.068,E2 -17622.068} C_VEL
LIN {X 0,Y 273.781,Z 316.372,A -85,B 0,C 180,E1 -17624.047,E2 -17624.047} C_VEL
LIN {X 0,Y 271.404,Z 316.678,A -85,B 0,C 180,E1 -17625.654,E2 -17625.654} C_VEL
LIN {X 0,Y 270.411,Z 316.795,A -85,B 0,C 180,E1 -17626.899,E2 -17626.899} C_VEL
LIN {X 0,Y 270.344,Z 316.798,A -85,B 0,C 180,E1 -17627.321,E2 -17627.321} C_VEL
LIN {X 0,Y 270.514,Z 316.787,A -85,B 0,C 180,E1 -17631.032,E2 -17631.032} C_VEL
LIN {X 0,Y 270.505,Z 316.779,A -85,B 0,C 180,E1 -17634.035,E2 -17634.035} C_VEL
LIN {X 0,Y 270.773,Z 316.741,A -85,B 0,C 180,E1 -17638.513,E2 -17638.513} C_VEL
LIN {X 0,Y 270.774,Z 316.753,A -85,B 0,C 180,E1 -17641.488,E2 -17641.488} C_VEL
LIN {X 0,Y 270.598,Z 316.769,A -85,B 0,C 180,E1 -17647.462,E2 -17647.462} C_VEL
LIN {X 0,Y 270.429,Z 316.795,A -85,B 0,C 180,E1 -17650.482,E2 -17650.482} C_VEL
LIN {X 0,Y 270.391,Z 316.795,A -85,B 0,C 180,E1 -17655.066,E2 -17655.066} C_VEL
LIN {X 0,Y 270.29,Z 316.808,A -85,B 0,C 180,E1 -17659.757,E2 -17659.757} C_VEL
LIN {X 0,Y 270.263,Z 316.812,A -85,B 0,C 180,E1 -17664.587,E2 -17664.587} C_VEL
LIN {X 0,Y 270.262,Z 316.808,A -85,B 0,C 180,E1 -17667.91,E2 -17667.91} C_VEL
LIN {X 0,Y 270.175,Z 316.825,A -85,B 0,C 180,E1 -17671.35,E2 -17671.35} C_VEL
LIN {X 0,Y 270.207,Z 316.827,A -85,B 0,C 180,E1 -17674.905,E2 -17674.905} C_VEL
LIN {X 0,Y 270.214,Z 316.824,A -85,B 0,C 180,E1 -17678.719,E2 -17678.719} C_VEL
LIN {X 0,Y 270.194,Z 316.825,A -85,B 0,C 180,E1 -17682.554,E2 -17682.554} C_VEL
LIN {X 0,Y 270.209,Z 316.81,A -85,B 0,C 180,E1 -17686.742,E2 -17686.742} C_VEL
LIN {X 0,Y 270.279,Z 316.942,A -85,B 0,C 180,E1 -17689.027,E2 -17689.027} C_VEL
LIN {X 0,Y 272.829,Z 326.071,A -85,B 0,C 180,E1 -17692.992,E2 -17692.992} C_VEL
LIN {X 0,Y 275.088,Z 335.014,A -85,B 0,C 180,E1 -17696.501,E2 -17696.501} C_VEL
LIN {X 0,Y 283.676,Z 352.318,A -85,B 0,C 180,E1 -17698.419,E2 -17698.419} C_VEL
LIN {X 0,Y 286.972,Z 360.044,A -85,B 0,C 180,E1 -17699.142,E2 -17699.142} C_VEL
LIN {X 0,Y 290.863,Z 381.745,A -85,B 0,C 180,E1 -17700.341,E2 -17700.341} C_VEL
LIN {X 0,Y 291.51,Z 387.881,A -85,B 0,C 180,E1 -17700.611,E2 -17700.611} C_VEL
LIN {X 0,Y 289.345,Z 444.543,A -85,B 0,C 180,E1 -17702.045,E2 -17702.045} C_VEL
LIN {X 0,Y 288.138,Z 458.007,A -85,B 0,C 180,E1 -17702.64,E2 -17702.64} C_VEL
LIN {X 0,Y 286.339,Z 471.003,A -85,B 0,C 180,E1 -17703.49,E2 -17703.49} C_VEL
LIN {X 0,Y 284.292,Z 482.776,A -85,B 0,C 180,E1 -17704.565,E2 -17704.565} C_VEL
LIN {X 0,Y 281.92,Z 494.122,A -85,B 0,C 180,E1 -17705.91,E2 -17705.91} C_VEL
LIN {X 0,Y 279.539,Z 504.377,A -85,B 0,C 180,E1 -17707.458,E2 -17707.458} C_VEL
LIN {X 0,Y 277.123,Z 513.622,A -85,B 0,C 180,E1 -17709.206,E2 -17709.206} C_VEL
LIN {X 0,Y 274.889,Z 521.617,A -85,B 0,C 180,E1 -17711.08,E2 -17711.08} C_VEL
LIN {X 0,Y 273.156,Z 528.758,A -85,B 0,C 180,E1 -17713.177,E2 -17713.177} C_VEL
LIN {X 0,Y 271.041,Z 535.731,A -85,B 0,C 180,E1 -17715.742,E2 -17715.742} C_VEL
LIN {X 0,Y 269.784,Z 540.368,A -85,B 0,C 180,E1 -17717.974,E2 -17717.974} C_VEL
LIN {X 0,Y 268.971,Z 543.924,A -85,B 0,C 180,E1 -17720.224,E2 -17720.224} C_VEL
LIN {X 0,Y 268.419,Z 546.498,A -85,B 0,C 180,E1 -17722.48,E2 -17722.48} C_VEL
LIN {X 0,Y 268.209,Z 548.135,A -85,B 0,C 180,E1 -17724.707,E2 -17724.707} C_VEL
LIN {X 0,Y 268.193,Z 548.919,A -85,B 0,C 180,E1 -17726.998,E2 -17726.998} C_VEL
LIN {X 0,Y 268.215,Z 548.935,A -85,B 0,C 180,E1 -17728.501,E2 -17728.501} C_VEL
LIN {X 0,Y 268.253,Z 548.565,A -85,B 0,C 180,E1 -17730.002,E2 -17730.002} C_VEL
LIN {X 0,Y 268.24,Z 547.762,A -85,B 0,C 180,E1 -17731.504,E2 -17731.504} C_VEL
LIN {X 0,Y 268.258,Z 546.536,A -85,B 0,C 180,E1 -17733.006,E2 -17733.006} C_VEL
LIN {X 0,Y 268.257,Z 543.707,A -85,B 0,C 180,E1 -17735.401,E2 -17735.401} C_VEL
LIN {X 0,Y 268.443,Z 540.233,A -85,B 0,C 180,E1 -17737.524,E2 -17737.524} C_VEL
LIN {X 0,Y 268.814,Z 535.419,A -85,B 0,C 180,E1 -17739.786,E2 -17739.786} C_VEL
LIN {X 0,Y 269.43,Z 529.314,A -85,B 0,C 180,E1 -17742.047,E2 -17742.047} C_VEL
LIN {X 0,Y 270.56,Z 521.719,A -85,B 0,C 180,E1 -17744.289,E2 -17744.289} C_VEL
LIN {X 0,Y 271.736,Z 513.947,A -85,B 0,C 180,E1 -17746.145,E2 -17746.145} C_VEL
LIN {X 0,Y 272.983,Z 504.429,A -85,B 0,C 180,E1 -17747.998,E2 -17747.998} C_VEL
LIN {X 0,Y 274.313,Z 493.829,A -85,B 0,C 180,E1 -17749.652,E2 -17749.652} C_VEL
LIN {X 0,Y 275.96,Z 482.081,A -85,B 0,C 180,E1 -17751.086,E2 -17751.086} C_VEL
LIN {X 0,Y 277.212,Z 470.637,A -85,B 0,C 180,E1 -17752.157,E2 -17752.157} C_VEL
LIN {X 0,Y 278.448,Z 457,A -85,B 0,C 180,E1 -17753.081,E2 -17753.081} C_VEL
LIN {X 0,Y 279.217,Z 444.245,A -85,B 0,C 180,E1 -17753.652,E2 -17753.652} C_VEL
LIN {X 0,Y 280.789,Z 383.399,A -85,B 0,C 180,E1 -17755.211,E2 -17755.211} C_VEL
LIN {X 0,Y 275.484,Z 342.171,A -85,B 0,C 180,E1 -17756.759,E2 -17756.759} C_VEL
LIN {X 0,Y 274.291,Z 336.705,A -85,B 0,C 180,E1 -17757.011,E2 -17757.011} C_VEL
LIN {X 0,Y 274.199,Z 336.24,A -85,B 0,C 180,E1 -17757.056,E2 -17757.056} C_VEL
LIN {X 0,Y 272.293,Z 326.46,A -85,B 0,C 180,E1 -17760.221,E2 -17760.221} C_VEL
LIN {X 0,Y 270.21,Z 316.822,A -85,B 0,C 180,E1 -17763.534,E2 -17763.534} C_VEL
LIN {X 0,Y 270.224,Z 316.826,A -85,B 0,C 180,E1 -17766.742,E2 -17766.742} C_VEL
LIN {X 0,Y 270.176,Z 316.83,A -85,B 0,C 180,E1 -17771.029,E2 -17771.029} C_VEL
LIN {X 0,Y 270.159,Z 316.831,A -85,B 0,C 180,E1 -17775.381,E2 -17775.381} C_VEL
LIN {X 0,Y 270.181,Z 316.826,A -85,B 0,C 180,E1 -17779.435,E2 -17779.435} C_VEL
LIN {X 0,Y 270.232,Z 316.82,A -85,B 0,C 180,E1 -17783.731,E2 -17783.731} C_VEL
LIN {X 0,Y 270.211,Z 316.825,A -85,B 0,C 180,E1 -17786.893,E2 -17786.893} C_VEL
LIN {X 0,Y 270.237,Z 316.817,A -85,B 0,C 180,E1 -17790.387,E2 -17790.387} C_VEL
LIN {X 0,Y 270.271,Z 316.817,A -85,B 0,C 180,E1 -17793.764,E2 -17793.764} C_VEL
LIN {X 0,Y 270.216,Z 316.826,A -85,B 0,C 180,E1 -17797.037,E2 -17797.037} C_VEL
LIN {X 0,Y 270.259,Z 316.811,A -85,B 0,C 180,E1 -17800.241,E2 -17800.241} C_VEL
LIN {X 0,Y 270.376,Z 316.8,A -85,B 0,C 180,E1 -17804.933,E2 -17804.933} C_VEL
LIN {X 0,Y 270.42,Z 316.8,A -85,B 0,C 180,E1 -17809.518,E2 -17809.518} C_VEL
LIN {X 0,Y 270.57,Z 316.766,A -85,B 0,C 180,E1 -17812.537,E2 -17812.537} C_VEL
LIN {X 0,Y 270.792,Z 316.752,A -85,B 0,C 180,E1 -17818.512,E2 -17818.512} C_VEL
LIN {X 0,Y 270.792,Z 316.75,A -85,B 0,C 180,E1 -17821.487,E2 -17821.487} C_VEL
LIN {X 0,Y 270.591,Z 316.766,A -85,B 0,C 180,E1 -17827.461,E2 -17827.461} C_VEL
LIN {X 0,Y 270.417,Z 316.8,A -85,B 0,C 180,E1 -17830.482,E2 -17830.482} C_VEL
LIN {X 0,Y 270.375,Z 316.801,A -85,B 0,C 180,E1 -17835.066,E2 -17835.066} C_VEL
LIN {X 0,Y 270.258,Z 316.818,A -85,B 0,C 180,E1 -17839.759,E2 -17839.759} C_VEL
LIN {X 0,Y 270.244,Z 316.82,A -85,B 0,C 180,E1 -17844.588,E2 -17844.588} C_VEL
LIN {X 0,Y 270.278,Z 316.812,A -85,B 0,C 180,E1 -17847.908,E2 -17847.908} C_VEL
LIN {X 0,Y 270.19,Z 316.828,A -85,B 0,C 180,E1 -17851.347,E2 -17851.347} C_VEL
LIN {X 0,Y 270.207,Z 316.823,A -85,B 0,C 180,E1 -17854.904,E2 -17854.904} C_VEL
LIN {X 0,Y 270.203,Z 316.823,A -85,B 0,C 180,E1 -17858.709,E2 -17858.709} C_VEL
LIN {X 0,Y 270.184,Z 316.825,A -85,B 0,C 180,E1 -17862.556,E2 -17862.556} C_VEL
LIN {X 0,Y 270.17,Z 316.827,A -85,B 0,C 180,E1 -17866.75,E2 -17866.75} C_VEL
LIN {X 0,Y 270.179,Z 316.829,A -85,B 0,C 180,E1 -17869.433,E2 -17869.433} C_VEL
LIN {X 0,Y 270.231,Z 316.825,A -85,B 0,C 180,E1 -17873.728,E2 -17873.728} C_VEL
LIN {X 0,Y 270.207,Z 316.825,A -85,B 0,C 180,E1 -17876.891,E2 -17876.891} C_VEL
LIN {X 0,Y 270.199,Z 316.828,A -85,B 0,C 180,E1 -17880.381,E2 -17880.381} C_VEL
LIN {X 0,Y 270.266,Z 316.819,A -85,B 0,C 180,E1 -17883.762,E2 -17883.762} C_VEL
LIN {X 0,Y 270.241,Z 316.821,A -85,B 0,C 180,E1 -17887.037,E2 -17887.037} C_VEL
LIN {X 0,Y 270.306,Z 316.813,A -85,B 0,C 180,E1 -17890.243,E2 -17890.243} C_VEL
LIN {X 0,Y 270.405,Z 316.802,A -85,B 0,C 180,E1 -17894.933,E2 -17894.933} C_VEL
LIN {X 0,Y 270.396,Z 316.828,A -85,B 0,C 180,E1 -17897.33,E2 -17897.33} C_VEL
LIN {X 0,Y 270.74,Z 318.287,A -85,B 0,C 180,E1 -17897.767,E2 -17897.767} C_VEL
LIN {X 0,Y 278.895,Z 340.46,A -85,B 0,C 180,E1 -17899.072,E2 -17899.072} C_VEL
LIN {X 0,Y 281.067,Z 348.092,A -85,B 0,C 180,E1 -17899.453,E2 -17899.453} C_VEL
LIN {X 0,Y 281.48,Z 351.473,A -85,B 0,C 180,E1 -17899.577,E2 -17899.577} C_VEL
LIN {X 0,Y 279.365,Z 425.216,A -85,B 0,C 180,E1 -17901.453,E2 -17901.453} C_VEL
LIN {X 0,Y 278.629,Z 438.43,A -85,B 0,C 180,E1 -17902.069,E2 -17902.069} C_VEL
LIN {X 0,Y 277.736,Z 451.624,A -85,B 0,C 180,E1 -17903.003,E2 -17903.003} C_VEL
LIN {X 0,Y 276.52,Z 463.586,A -85,B 0,C 180,E1 -17904.163,E2 -17904.163} C_VEL
LIN {X 0,Y 275.213,Z 475.02,A -85,B 0,C 180,E1 -17905.604,E2 -17905.604} C_VEL
LIN {X 0,Y 273.755,Z 485.368,A -85,B 0,C 180,E1 -17907.239,E2 -17907.239} C_VEL
LIN {X 0,Y 272.522,Z 493.814,A -85,B 0,C 180,E1 -17908.89,E2 -17908.89} C_VEL
LIN {X 0,Y 271.11,Z 502.97,A -85,B 0,C 180,E1 -17911.112,E2 -17911.112} C_VEL
LIN {X 0,Y 270.073,Z 510.337,A -85,B 0,C 180,E1 -17913.354,E2 -17913.354} C_VEL
LIN {X 0,Y 269.42,Z 515.326,A -85,B 0,C 180,E1 -17915.236,E2 -17915.236} C_VEL
LIN {X 0,Y 268.865,Z 520.171,A -85,B 0,C 180,E1 -17917.508,E2 -17917.508} C_VEL
LIN {X 0,Y 268.403,Z 523.901,A -85,B 0,C 180,E1 -17919.797,E2 -17919.797} C_VEL
LIN {X 0,Y 268.125,Z 526.592,A -85,B 0,C 180,E1 -17922.102,E2 -17922.102} C_VEL
LIN {X 0,Y 268.068,Z 528.11,A -85,B 0,C 180,E1 -17924.062,E2 -17924.062} C_VEL
LIN {X 0,Y 268.039,Z 529.076,A -85,B 0,C 180,E1 -17926.761,E2 -17926.761} C_VEL
LIN {X 0,Y 268.401,Z 528.777,A -85,B 0,C 180,E1 -17929.499,E2 -17929.499} C_VEL
LIN {X 0,Y 268.788,Z 527.749,A -85,B 0,C 180,E1 -17931.47,E2 -17931.47} C_VEL
LIN {X 0,Y 269.753,Z 525.129,A -85,B 0,C 180,E1 -17934.236,E2 -17934.236} C_VEL
LIN {X 0,Y 271.07,Z 521.083,A -85,B 0,C 180,E1 -17936.98,E2 -17936.98} C_VEL
LIN {X 0,Y 272.566,Z 516.261,A -85,B 0,C 180,E1 -17939.331,E2 -17939.331} C_VEL
LIN {X 0,Y 274.471,Z 510.059,A -85,B 0,C 180,E1 -17941.66,E2 -17941.66} C_VEL
LIN {X 0,Y 276.749,Z 502.239,A -85,B 0,C 180,E1 -17943.962,E2 -17943.962} C_VEL
LIN {X 0,Y 279.16,Z 493.319,A -85,B 0,C 180,E1 -17946.021,E2 -17946.021} C_VEL
LIN {X 0,Y 281.38,Z 484.099,A -85,B 0,C 180,E1 -17947.726,E2 -17947.726} C_VEL
LIN {X 0,Y 283.89,Z 472.849,A -85,B 0,C 180,E1 -17949.37,E2 -17949.37} C_VEL
LIN {X 0,Y 285.968,Z 461.369,A -85,B 0,C 180,E1 -17950.673,E2 -17950.673} C_VEL
LIN {X 0,Y 287.716,Z 449.224,A -85,B 0,C 180,E1 -17951.727,E2 -17951.727} C_VEL
LIN {X 0,Y 289.145,Z 436.38,A -85,B 0,C 180,E1 -17952.529,E2 -17952.529} C_VEL
LIN {X 0,Y 290.024,Z 424.303,A -85,B 0,C 180,E1 -17953.02,E2 -17953.02} C_VEL
LIN {X 0,Y 292.465,Z 360.629,A -85,B 0,C 180,E1 -17954.606,E2 -17954.606} C_VEL
LIN {X 0,Y 286.263,Z 347.036,A -85,B 0,C 180,E1 -17955.898,E2 -17955.898} C_VEL
LIN {X 0,Y 279.634,Z 334.333,A -85,B 0,C 180,E1 -17957.315,E2 -17957.315} C_VEL
LIN {X 0,Y 274.821,Z 326.115,A -85,B 0,C 180,E1 -17958.375,E2 -17958.375} C_VEL
LIN {X 0,Y 270.906,Z 319.375,A -85,B 0,C 180,E1 -17959.279,E2 -17959.279} C_VEL
LIN {X 0,Y 270.173,Z 316.872,A -85,B 0,C 180,E1 -17960.318,E2 -17960.318} C_VEL
LIN {X 0,Y 270.206,Z 316.808,A -85,B 0,C 180,E1 -17963.732,E2 -17963.732} C_VEL
LIN {X 0,Y 270.189,Z 316.831,A -85,B 0,C 180,E1 -17966.891,E2 -17966.891} C_VEL
LIN {X 0,Y 270.17,Z 316.832,A -85,B 0,C 180,E1 -17970.38,E2 -17970.38} C_VEL
LIN {X 0,Y 270.189,Z 316.83,A -85,B 0,C 180,E1 -17973.756,E2 -17973.756} C_VEL
LIN {X 0,Y 270.191,Z 316.829,A -85,B 0,C 180,E1 -17977.035,E2 -17977.035} C_VEL
LIN {X 0,Y 270.26,Z 316.813,A -85,B 0,C 180,E1 -17980.848,E2 -17980.848} C_VEL
LIN {X 0,Y 270.39,Z 316.803,A -85,B 0,C 180,E1 -17984.935,E2 -17984.935} C_VEL
LIN {X 0,Y 270.344,Z 316.798,A -85,B 0,C 180,E1 -17987.321,E2 -17987.321} C_VEL
LIN {X 0,Y 269.752,Z 316.873,A -85,B 0,C 180,E1 -17988.565,E2 -17988.565} C_VEL
LIN {X 0,Y 267.057,Z 317.22,A -85,B 0,C 180,E1 -17990.597,E2 -17990.597} C_VEL
LIN {X 0,Y 263.857,Z 317.607,A -85,B 0,C 180,E1 -17993.093,E2 -17993.093} C_VEL
LIN {X 0,Y 263.465,Z 317.654,A -85,B 0,C 180,E1 -17993.955,E2 -17993.955} C_VEL
LIN {X 0,Y 263.738,Z 317.617,A -85,B 0,C 180,E1 -17998.473,E2 -17998.473} C_VEL
LIN {X 0,Y 263.739,Z 317.629,A -85,B 0,C 180,E1 -18001.527,E2 -18001.527} C_VEL
LIN {X 0,Y 263.56,Z 317.643,A -85,B 0,C 180,E1 -18007.662,E2 -18007.662} C_VEL
LIN {X 0,Y 263.362,Z 317.678,A -85,B 0,C 180,E1 -18010.766,E2 -18010.766} C_VEL
LIN {X 0,Y 263.339,Z 317.679,A -85,B 0,C 180,E1 -18015.479,E2 -18015.479} C_VEL
LIN {X 0,Y 263.252,Z 317.689,A -85,B 0,C 180,E1 -18020.308,E2 -18020.308} C_VEL
LIN {X 0,Y 263.199,Z 317.698,A -85,B 0,C 180,E1 -18025.293,E2 -18025.293} C_VEL
LIN {X 0,Y 263.17,Z 317.693,A -85,B 0,C 180,E1 -18028.731,E2 -18028.731} C_VEL
LIN {X 0,Y 263.124,Z 317.7,A -85,B 0,C 180,E1 -18032.29,E2 -18032.29} C_VEL
LIN {X 0,Y 263.181,Z 317.697,A -85,B 0,C 180,E1 -18035.98,E2 -18035.98} C_VEL
LIN {X 0,Y 263.146,Z 317.705,A -85,B 0,C 180,E1 -18039.866,E2 -18039.866} C_VEL
LIN {X 0,Y 263.136,Z 317.707,A -85,B 0,C 180,E1 -18043.982,E2 -18043.982} C_VEL
LIN {X 0,Y 263.206,Z 317.74,A -85,B 0,C 180,E1 -18047.869,E2 -18047.869} C_VEL
LIN {X 0,Y 265.72,Z 326.544,A -85,B 0,C 180,E1 -18051.892,E2 -18051.892} C_VEL
LIN {X 0,Y 267.73,Z 334.453,A -85,B 0,C 180,E1 -18055.199,E2 -18055.199} C_VEL
LIN {X 0,Y 269.892,Z 338.738,A -85,B 0,C 180,E1 -18055.742,E2 -18055.742} C_VEL
LIN {X 0,Y 275.385,Z 349.505,A -85,B 0,C 180,E1 -18057.031,E2 -18057.031} C_VEL
LIN {X 0,Y 281.389,Z 362.356,A -85,B 0,C 180,E1 -18058.391,E2 -18058.391} C_VEL
LIN {X 0,Y 285.16,Z 383.806,A -85,B 0,C 180,E1 -18059.611,E2 -18059.611} C_VEL
LIN {X 0,Y 285.663,Z 389.11,A -85,B 0,C 180,E1 -18059.844,E2 -18059.844} C_VEL
LIN {X 0,Y 283.442,Z 444.078,A -85,B 0,C 180,E1 -18061.254,E2 -18061.254} C_VEL
LIN {X 0,Y 282.265,Z 456.901,A -85,B 0,C 180,E1 -18061.819,E2 -18061.819} C_VEL
LIN {X 0,Y 280.406,Z 470.128,A -85,B 0,C 180,E1 -18062.682,E2 -18062.682} C_VEL
LIN {X 0,Y 278.259,Z 482.057,A -85,B 0,C 180,E1 -18063.771,E2 -18063.771} C_VEL
LIN {X 0,Y 275.81,Z 493.475,A -85,B 0,C 180,E1 -18065.14,E2 -18065.14} C_VEL
LIN {X 0,Y 273.251,Z 503.793,A -85,B 0,C 180,E1 -18066.709,E2 -18066.709} C_VEL
LIN {X 0,Y 270.998,Z 512.249,A -85,B 0,C 180,E1 -18068.314,E2 -18068.314} C_VEL
LIN {X 0,Y 268.353,Z 521.213,A -85,B 0,C 180,E1 -18070.423,E2 -18070.423} C_VEL
LIN {X 0,Y 266.341,Z 528.878,A -85,B 0,C 180,E1 -18072.734,E2 -18072.734} C_VEL
LIN {X 0,Y 264.159,Z 535.767,A -85,B 0,C 180,E1 -18075.362,E2 -18075.362} C_VEL
LIN {X 0,Y 262.802,Z 540.338,A -85,B 0,C 180,E1 -18077.649,E2 -18077.649} C_VEL
LIN {X 0,Y 261.95,Z 543.841,A -85,B 0,C 180,E1 -18079.959,E2 -18079.959} C_VEL
LIN {X 0,Y 261.355,Z 546.357,A -85,B 0,C 180,E1 -18082.275,E2 -18082.275} C_VEL
LIN {X 0,Y 261.124,Z 548.052,A -85,B 0,C 180,E1 -18084.772,E2 -18084.772} C_VEL
LIN {X 0,Y 261.106,Z 548.667,A -85,B 0,C 180,E1 -18086.916,E2 -18086.916} C_VEL
LIN {X 0,Y 261.141,Z 548.657,A -85,B 0,C 180,E1 -18088.46,E2 -18088.46} C_VEL
LIN {X 0,Y 261.176,Z 548.251,A -85,B 0,C 180,E1 -18090.002,E2 -18090.002} C_VEL
LIN {X 0,Y 261.167,Z 547.403,A -85,B 0,C 180,E1 -18091.544,E2 -18091.544} C_VEL
LIN {X 0,Y 261.166,Z 546.148,A -85,B 0,C 180,E1 -18093.087,E2 -18093.087} C_VEL
LIN {X 0,Y 261.167,Z 543.565,A -85,B 0,C 180,E1 -18095.329,E2 -18095.329} C_VEL
LIN {X 0,Y 261.365,Z 539.724,A -85,B 0,C 180,E1 -18097.729,E2 -18097.729} C_VEL
LIN {X 0,Y 261.767,Z 534.842,A -85,B 0,C 180,E1 -18100.053,E2 -18100.053} C_VEL
LIN {X 0,Y 262.444,Z 528.663,A -85,B 0,C 180,E1 -18102.373,E2 -18102.373} C_VEL
LIN {X 0,Y 263.636,Z 520.979,A -85,B 0,C 180,E1 -18104.672,E2 -18104.672} C_VEL
LIN {X 0,Y 264.853,Z 513.091,A -85,B 0,C 180,E1 -18106.576,E2 -18106.576} C_VEL
LIN {X 0,Y 266.183,Z 503.411,A -85,B 0,C 180,E1 -18108.474,E2 -18108.474} C_VEL
LIN {X 0,Y 267.644,Z 492.664,A -85,B 0,C 180,E1 -18110.162,E2 -18110.162} C_VEL
LIN {X 0,Y 269.074,Z 482.301,A -85,B 0,C 180,E1 -18111.451,E2 -18111.451} C_VEL
LIN {X 0,Y 270.509,Z 469.928,A -85,B 0,C 180,E1 -18112.636,E2 -18112.636} C_VEL
LIN {X 0,Y 271.708,Z 456.897,A -85,B 0,C 180,E1 -18113.537,E2 -18113.537} C_VEL
LIN {X 0,Y 272.494,Z 444.245,A -85,B 0,C 180,E1 -18114.121,E2 -18114.121} C_VEL
LIN {X 0,Y 274.115,Z 383.79,A -85,B 0,C 180,E1 -18115.709,E2 -18115.709} C_VEL
LIN {X 0,Y 268.678,Z 341.562,A -85,B 0,C 180,E1 -18117.348,E2 -18117.348} C_VEL
LIN {X 0,Y 266.975,Z 335.876,A -85,B 0,C 180,E1 -18117.707,E2 -18117.707} C_VEL
LIN {X 0,Y 264.883,Z 325.666,A -85,B 0,C 180,E1 -18121.134,E2 -18121.134} C_VEL
LIN {X 0,Y 263.18,Z 317.7,A -85,B 0,C 180,E1 -18123.982,E2 -18123.982} C_VEL
LIN {X 0,Y 263.166,Z 317.704,A -85,B 0,C 180,E1 -18127.898,E2 -18127.898} C_VEL
LIN {X 0,Y 263.131,Z 317.708,A -85,B 0,C 180,E1 -18131.894,E2 -18131.894} C_VEL
LIN {X 0,Y 263.112,Z 317.71,A -85,B 0,C 180,E1 -18136.156,E2 -18136.156} C_VEL
LIN {X 0,Y 263.113,Z 317.707,A -85,B 0,C 180,E1 -18140.128,E2 -18140.128} C_VEL
LIN {X 0,Y 263.17,Z 317.7,A -85,B 0,C 180,E1 -18144.019,E2 -18144.019} C_VEL
LIN {X 0,Y 263.141,Z 317.704,A -85,B 0,C 180,E1 -18147.712,E2 -18147.712} C_VEL
LIN {X 0,Y 263.21,Z 317.696,A -85,B 0,C 180,E1 -18151.783,E2 -18151.783} C_VEL
LIN {X 0,Y 263.209,Z 317.7,A -85,B 0,C 180,E1 -18155.212,E2 -18155.212} C_VEL
LIN {X 0,Y 263.243,Z 317.688,A -85,B 0,C 180,E1 -18159.691,E2 -18159.691} C_VEL
LIN {X 0,Y 263.318,Z 317.679,A -85,B 0,C 180,E1 -18164.52,E2 -18164.52} C_VEL
LIN {X 0,Y 263.362,Z 317.677,A -85,B 0,C 180,E1 -18169.234,E2 -18169.234} C_VEL
LIN {X 0,Y 263.534,Z 317.642,A -85,B 0,C 180,E1 -18172.337,E2 -18172.337} C_VEL
LIN {X 0,Y 263.756,Z 317.628,A -85,B 0,C 180,E1 -18178.473,E2 -18178.473} C_VEL
LIN {X 0,Y 263.757,Z 317.626,A -85,B 0,C 180,E1 -18181.527,E2 -18181.527} C_VEL
LIN {X 0,Y 263.551,Z 317.642,A -85,B 0,C 180,E1 -18187.662,E2 -18187.662} C_VEL
LIN {X 0,Y 263.36,Z 317.679,A -85,B 0,C 180,E1 -18190.766,E2 -18190.766} C_VEL
LIN {X 0,Y 263.317,Z 317.678,A -85,B 0,C 180,E1 -18195.48,E2 -18195.48} C_VEL
LIN {X 0,Y 263.242,Z 317.693,A -85,B 0,C 180,E1 -18200.308,E2 -18200.308} C_VEL
LIN {X 0,Y 263.199,Z 317.699,A -85,B 0,C 180,E1 -18205.292,E2 -18205.292} C_VEL
LIN {X 0,Y 263.185,Z 317.698,A -85,B 0,C 180,E1 -18208.729,E2 -18208.729} C_VEL
LIN {X 0,Y 263.139,Z 317.703,A -85,B 0,C 180,E1 -18212.287,E2 -18212.287} C_VEL
LIN {X 0,Y 263.187,Z 317.697,A -85,B 0,C 180,E1 -18216.762,E2 -18216.762} C_VEL
LIN {X 0,Y 263.135,Z 317.706,A -85,B 0,C 180,E1 -18221.593,E2 -18221.593} C_VEL
LIN {X 0,Y 263.129,Z 317.705,A -85,B 0,C 180,E1 -18223.983,E2 -18223.983} C_VEL
LIN {X 0,Y 263.129,Z 317.705,A -85,B 0,C 180,E1 -18228.405,E2 -18228.405} C_VEL
LIN {X 0,Y 263.189,Z 317.699,A -85,B 0,C 180,E1 -18233.235,E2 -18233.235} C_VEL
LIN {X 0,Y 263.137,Z 317.708,A -85,B 0,C 180,E1 -18237.71,E2 -18237.71} C_VEL
LIN {X 0,Y 263.2,Z 317.699,A -85,B 0,C 180,E1 -18241.783,E2 -18241.783} C_VEL
LIN {X 0,Y 263.229,Z 317.694,A -85,B 0,C 180,E1 -18245.198,E2 -18245.198} C_VEL
LIN {X 0,Y 263.272,Z 317.687,A -85,B 0,C 180,E1 -18249.692,E2 -18249.692} C_VEL
LIN {X 0,Y 263.354,Z 317.681,A -85,B 0,C 180,E1 -18254.52,E2 -18254.52} C_VEL
LIN {X 0,Y 263.363,Z 317.772,A -85,B 0,C 180,E1 -18256.928,E2 -18256.928} C_VEL
LIN {X 0,Y 263.468,Z 318.247,A -85,B 0,C 180,E1 -18257.104,E2 -18257.104} C_VEL
LIN {X 0,Y 272.183,Z 341.593,A -85,B 0,C 180,E1 -18258.552,E2 -18258.552} C_VEL
LIN {X 0,Y 274.544,Z 349.719,A -85,B 0,C 180,E1 -18258.976,E2 -18258.976} C_VEL
LIN {X 0,Y 274.795,Z 353.518,A -85,B 0,C 180,E1 -18259.103,E2 -18259.103} C_VEL
LIN {X 0,Y 272.624,Z 426.188,A -85,B 0,C 180,E1 -18261.004,E2 -18261.004} C_VEL
LIN {X 0,Y 271.837,Z 439.943,A -85,B 0,C 180,E1 -18261.683,E2 -18261.683} C_VEL
LIN {X 0,Y 270.896,Z 452.746,A -85,B 0,C 180,E1 -18262.638,E2 -18262.638} C_VEL
LIN {X 0,Y 269.634,Z 464.509,A -85,B 0,C 180,E1 -18263.826,E2 -18263.826} C_VEL
LIN {X 0,Y 268.269,Z 475.827,A -85,B 0,C 180,E1 -18265.302,E2 -18265.302} C_VEL
LIN {X 0,Y 266.785,Z 486.056,A -85,B 0,C 180,E1 -18266.978,E2 -18266.978} C_VEL
LIN {X 0,Y 265.382,Z 495.245,A -85,B 0,C 180,E1 -18268.86,E2 -18268.86} C_VEL
LIN {X 0,Y 263.968,Z 504.2,A -85,B 0,C 180,E1 -18271.142,E2 -18271.142} C_VEL
LIN {X 0,Y 262.905,Z 511.389,A -85,B 0,C 180,E1 -18273.446,E2 -18273.446} C_VEL
LIN {X 0,Y 262.113,Z 517.918,A -85,B 0,C 180,E1 -18276.155,E2 -18276.155} C_VEL
LIN {X 0,Y 261.568,Z 522.248,A -85,B 0,C 180,E1 -18278.496,E2 -18278.496} C_VEL
LIN {X 0,Y 261.124,Z 525.506,A -85,B 0,C 180,E1 -18280.857,E2 -18280.857} C_VEL
LIN {X 0,Y 261.014,Z 527.124,A -85,B 0,C 180,E1 -18282.437,E2 -18282.437} C_VEL
LIN {X 0,Y 260.964,Z 528.384,A -85,B 0,C 180,E1 -18284.185,E2 -18284.185} C_VEL
LIN {X 0,Y 260.973,Z 529.378,A -85,B 0,C 180,E1 -18287.229,E2 -18287.229} C_VEL
LIN {X 0,Y 261.34,Z 529.049,A -85,B 0,C 180,E1 -18289.742,E2 -18289.742} C_VEL
LIN {X 0,Y 261.87,Z 527.813,A -85,B 0,C 180,E1 -18292.067,E2 -18292.067} C_VEL
LIN {X 0,Y 262.799,Z 525.42,A -85,B 0,C 180,E1 -18294.598,E2 -18294.598} C_VEL
LIN {X 0,Y 263.927,Z 522.195,A -85,B 0,C 180,E1 -18296.913,E2 -18296.913} C_VEL
LIN {X 0,Y 265.514,Z 517.451,A -85,B 0,C 180,E1 -18299.427,E2 -18299.427} C_VEL
LIN {X 0,Y 267.38,Z 511.81,A -85,B 0,C 180,E1 -18301.712,E2 -18301.712} C_VEL
LIN {X 0,Y 269.684,Z 504.329,A -85,B 0,C 180,E1 -18304.073,E2 -18304.073} C_VEL
LIN {X 0,Y 271.956,Z 496.634,A -85,B 0,C 180,E1 -18306.006,E2 -18306.006} C_VEL
LIN {X 0,Y 274.446,Z 487.202,A -85,B 0,C 180,E1 -18307.919,E2 -18307.919} C_VEL
LIN {X 0,Y 276.979,Z 476.652,A -85,B 0,C 180,E1 -18309.603,E2 -18309.603} C_VEL
LIN {X 0,Y 279.306,Z 465.066,A -85,B 0,C 180,E1 -18311.05,E2 -18311.05} C_VEL
LIN {X 0,Y 281.165,Z 453.469,A -85,B 0,C 180,E1 -18312.176,E2 -18312.176} C_VEL
LIN {X 0,Y 282.67,Z 441.843,A -85,B 0,C 180,E1 -18313.01,E2 -18313.01} C_VEL
LIN {X 0,Y 283.787,Z 428.912,A -85,B 0,C 180,E1 -18313.652,E2 -18313.652} C_VEL
LIN {X 0,Y 284.837,Z 408.99,A -85,B 0,C 180,E1 -18314.199,E2 -18314.199} C_VEL
LIN {X 0,Y 286.614,Z 362.728,A -85,B 0,C 180,E1 -18315.364,E2 -18315.364} C_VEL
LIN {X 0,Y 279.95,Z 348.191,A -85,B 0,C 180,E1 -18316.817,E2 -18316.817} C_VEL
LIN {X 0,Y 271.276,Z 332.193,A -85,B 0,C 180,E1 -18318.775,E2 -18318.775} C_VEL
LIN {X 0,Y 265.674,Z 323.082,A -85,B 0,C 180,E1 -18320.098,E2 -18320.098} C_VEL
LIN {X 0,Y 263.563,Z 319.407,A -85,B 0,C 180,E1 -18320.646,E2 -18320.646} C_VEL
LIN {X 0,Y 263.126,Z 317.711,A -85,B 0,C 180,E1 -18321.528,E2 -18321.528} C_VEL
LIN {X 0,Y 263.144,Z 317.685,A -85,B 0,C 180,E1 -18324.015,E2 -18324.015} C_VEL
LIN {X 0,Y 263.116,Z 317.709,A -85,B 0,C 180,E1 -18327.71,E2 -18327.71} C_VEL
LIN {X 0,Y 263.135,Z 317.701,A -85,B 0,C 180,E1 -18331.804,E2 -18331.804} C_VEL
LIN {X 0,Y 263.177,Z 317.694,A -85,B 0,C 180,E1 -18335.217,E2 -18335.217} C_VEL
LIN {X 0,Y 263.25,Z 317.683,A -85,B 0,C 180,E1 -18339.693,E2 -18339.693} C_VEL
LIN {X 0,Y 263.338,Z 317.676,A -85,B 0,C 180,E1 -18344.522,E2 -18344.522} C_VEL
LIN {X 0,Y 263.342,Z 317.676,A -85,B 0,C 180,E1 -18349.233,E2 -18349.233} C_VEL
LIN {X 0,Y 263.516,Z 317.647,A -85,B 0,C 180,E1 -18352.337,E2 -18352.337} C_VEL
LIN {X 0,Y 263.465,Z 317.654,A -85,B 0,C 180,E1 -18353.955,E2 -18353.955} C_VEL
LIN {X 0,Y 262.727,Z 317.758,A -85,B 0,C 180,E1 -18355.233,E2 -18355.233} C_VEL
LIN {X 0,Y 260.009,Z 318.088,A -85,B 0,C 180,E1 -18357.324,E2 -18357.324} C_VEL
LIN {X 0,Y 257.009,Z 318.466,A -85,B 0,C 180,E1 -18359.893,E2 -18359.893} C_VEL
LIN {X 0,Y 256.703,Z 318.502,A -85,B 0,C 180,E1 -18360.778,E2 -18360.778} C_VEL
LIN {X 0,Y 256.474,Z 318.537,A -85,B 0,C 180,E1 -18366.293,E2 -18366.293} C_VEL
LIN {X 0,Y 256.449,Z 318.528,A -85,B 0,C 180,E1 -18369.464,E2 -18369.464} C_VEL
LIN {X 0,Y 256.242,Z 318.55,A -85,B 0,C 180,E1 -18374.291,E2 -18374.291} C_VEL
LIN {X 0,Y 256.199,Z 318.565,A -85,B 0,C 180,E1 -18377.563,E2 -18377.563} C_VEL
LIN {X 0,Y 256.146,Z 318.58,A -85,B 0,C 180,E1 -18381.121,E2 -18381.121} C_VEL
LIN {X 0,Y 256.178,Z 318.57,A -85,B 0,C 180,E1 -18385.14,E2 -18385.14} C_VEL
LIN {X 0,Y 256.104,Z 318.582,A -85,B 0,C 180,E1 -18389.601,E2 -18389.601} C_VEL
LIN {X 0,Y 256.076,Z 318.584,A -85,B 0,C 180,E1 -18393.292,E2 -18393.292} C_VEL
LIN {X 0,Y 256.133,Z 318.583,A -85,B 0,C 180,E1 -18397.281,E2 -18397.281} C_VEL
LIN {X 0,Y 256.077,Z 318.588,A -85,B 0,C 180,E1 -18401.199,E2 -18401.199} C_VEL
LIN {X 0,Y 256.07,Z 318.568,A -85,B 0,C 180,E1 -18405.528,E2 -18405.528} C_VEL
LIN {X 0,Y 256.132,Z 318.702,A -85,B 0,C 180,E1 -18406.692,E2 -18406.692} C_VEL
LIN {X 0,Y 258.353,Z 326.192,A -85,B 0,C 180,E1 -18410.322,E2 -18410.322} C_VEL
LIN {X 0,Y 260.475,Z 334.132,A -85,B 0,C 180,E1 -18413.845,E2 -18413.845} C_VEL
LIN {X 0,Y 262.91,Z 338.728,A -85,B 0,C 180,E1 -18414.48,E2 -18414.48} C_VEL
LIN {X 0,Y 269.097,Z 350.668,A -85,B 0,C 180,E1 -18416.014,E2 -18416.014} C_VEL
LIN {X 0,Y 275.638,Z 364.602,A -85,B 0,C 180,E1 -18417.569,E2 -18417.569} C_VEL
LIN {X 0,Y 276.559,Z 368.477,A -85,B 0,C 180,E1 -18417.842,E2 -18417.842} C_VEL
LIN {X 0,Y 279.725,Z 387.666,A -85,B 0,C 180,E1 -18418.94,E2 -18418.94} C_VEL
LIN {X 0,Y 279.718,Z 392.696,A -85,B 0,C 180,E1 -18419.098,E2 -18419.098} C_VEL
LIN {X 0,Y 277.542,Z 444.118,A -85,B 0,C 180,E1 -18420.446,E2 -18420.446} C_VEL
LIN {X 0,Y 276.257,Z 457.465,A -85,B 0,C 180,E1 -18421.056,E2 -18421.056} C_VEL
LIN {X 0,Y 274.356,Z 470.352,A -85,B 0,C 180,E1 -18421.923,E2 -18421.923} C_VEL
LIN {X 0,Y 272.27,Z 481.366,A -85,B 0,C 180,E1 -18422.941,E2 -18422.941} C_VEL
LIN {X 0,Y 270.045,Z 491.577,A -85,B 0,C 180,E1 -18424.159,E2 -18424.159} C_VEL
LIN {X 0,Y 267.314,Z 502.176,A -85,B 0,C 180,E1 -18425.748,E2 -18425.748} C_VEL
LIN {X 0,Y 264.436,Z 512.612,A -85,B 0,C 180,E1 -18427.748,E2 -18427.748} C_VEL
LIN {X 0,Y 261.586,Z 521.695,A -85,B 0,C 180,E1 -18429.975,E2 -18429.975} C_VEL
LIN {X 0,Y 259.541,Z 529.005,A -85,B 0,C 180,E1 -18432.267,E2 -18432.267} C_VEL
LIN {X 0,Y 257.294,Z 535.786,A -85,B 0,C 180,E1 -18434.963,E2 -18434.963} C_VEL
LIN {X 0,Y 255.831,Z 540.291,A -85,B 0,C 180,E1 -18437.307,E2 -18437.307} C_VEL
LIN {X 0,Y 255.177,Z 542.682,A -85,B 0,C 180,E1 -18438.887,E2 -18438.887} C_VEL
LIN {X 0,Y 254.313,Z 546.216,A -85,B 0,C 180,E1 -18442.06,E2 -18442.06} C_VEL
LIN {X 0,Y 253.994,Z 548.068,A -85,B 0,C 180,E1 -18445.241,E2 -18445.241} C_VEL
LIN {X 0,Y 254.02,Z 548.415,A -85,B 0,C 180,E1 -18446.83,E2 -18446.83} C_VEL
LIN {X 0,Y 254.068,Z 548.378,A -85,B 0,C 180,E1 -18448.417,E2 -18448.417} C_VEL
LIN {X 0,Y 254.102,Z 547.922,A -85,B 0,C 180,E1 -18450.002,E2 -18450.002} C_VEL
LIN {X 0,Y 254.094,Z 547.041,A -85,B 0,C 180,E1 -18451.587,E2 -18451.587} C_VEL
LIN {X 0,Y 254.078,Z 545.756,A -85,B 0,C 180,E1 -18453.174,E2 -18453.174} C_VEL
LIN {X 0,Y 254.088,Z 543.383,A -85,B 0,C 180,E1 -18455.28,E2 -18455.28} C_VEL
LIN {X 0,Y 254.316,Z 539.21,A -85,B 0,C 180,E1 -18457.945,E2 -18457.945} C_VEL
LIN {X 0,Y 254.739,Z 534.259,A -85,B 0,C 180,E1 -18460.333,E2 -18460.333} C_VEL
LIN {X 0,Y 255.457,Z 528.004,A -85,B 0,C 180,E1 -18462.717,E2 -18462.717} C_VEL
LIN {X 0,Y 256.688,Z 520.202,A -85,B 0,C 180,E1 -18465.079,E2 -18465.079} C_VEL
LIN {X 0,Y 257.971,Z 512.195,A -85,B 0,C 180,E1 -18467.032,E2 -18467.032} C_VEL
LIN {X 0,Y 259.435,Z 502.396,A -85,B 0,C 180,E1 -18468.972,E2 -18468.972} C_VEL
LIN {X 0,Y 260.748,Z 492.796,A -85,B 0,C 180,E1 -18470.514,E2 -18470.514} C_VEL
LIN {X 0,Y 262.227,Z 482.523,A -85,B 0,C 180,E1 -18471.833,E2 -18471.833} C_VEL
LIN {X 0,Y 263.69,Z 470.352,A -85,B 0,C 180,E1 -18473.047,E2 -18473.047} C_VEL
LIN {X 0,Y 264.972,Z 456.789,A -85,B 0,C 180,E1 -18474.017,E2 -18474.017} C_VEL
LIN {X 0,Y 265.782,Z 444.226,A -85,B 0,C 180,E1 -18474.614,E2 -18474.614} C_VEL
LIN {X 0,Y 267.436,Z 384.393,A -85,B 0,C 180,E1 -18476.227,E2 -18476.227} C_VEL
LIN {X 0,Y 262.407,Z 344.688,A -85,B 0,C 180,E1 -18477.811,E2 -18477.811} C_VEL
LIN {X 0,Y 261.446,Z 340.908,A -85,B 0,C 180,E1 -18478.009,E2 -18478.009} C_VEL
LIN {X 0,Y 259.697,Z 335.66,A -85,B 0,C 180,E1 -18478.353,E2 -18478.353} C_VEL
LIN {X 0,Y 257.424,Z 324.64,A -85,B 0,C 180,E1 -18482.184,E2 -18482.184} C_VEL
LIN {X 0,Y 256.11,Z 318.585,A -85,B 0,C 180,E1 -18484.446,E2 -18484.446} C_VEL
LIN {X 0,Y 256.122,Z 318.581,A -85,B 0,C 180,E1 -18487.272,E2 -18487.272} C_VEL
LIN {X 0,Y 256.062,Z 318.588,A -85,B 0,C 180,E1 -18491.205,E2 -18491.205} C_VEL
LIN {X 0,Y 256.048,Z 318.589,A -85,B 0,C 180,E1 -18495.535,E2 -18495.535} C_VEL
LIN {X 0,Y 256.062,Z 318.588,A -85,B 0,C 180,E1 -18498.797,E2 -18498.797} C_VEL
LIN {X 0,Y 256.137,Z 318.578,A -85,B 0,C 180,E1 -18502.868,E2 -18502.868} C_VEL
LIN {X 0,Y 256.076,Z 318.583,A -85,B 0,C 180,E1 -18506.708,E2 -18506.708} C_VEL
LIN {X 0,Y 256.122,Z 318.575,A -85,B 0,C 180,E1 -18510.401,E2 -18510.401} C_VEL
LIN {X 0,Y 256.179,Z 318.573,A -85,B 0,C 180,E1 -18514.87,E2 -18514.87} C_VEL
LIN {X 0,Y 256.156,Z 318.576,A -85,B 0,C 180,E1 -18519.104,E2 -18519.104} C_VEL
LIN {X 0,Y 256.238,Z 318.562,A -85,B 0,C 180,E1 -18524.081,E2 -18524.081} C_VEL
LIN {X 0,Y 256.296,Z 318.559,A -85,B 0,C 180,E1 -18527.328,E2 -18527.328} C_VEL
LIN {X 0,Y 256.442,Z 318.533,A -85,B 0,C 180,E1 -18530.623,E2 -18530.623} C_VEL
LIN {X 0,Y 256.466,Z 318.522,A -85,B 0,C 180,E1 -18533.707,E2 -18533.707} C_VEL
LIN {X 0,Y 256.719,Z 318.505,A -85,B 0,C 180,E1 -18538.431,E2 -18538.431} C_VEL
LIN {X 0,Y 256.72,Z 318.503,A -85,B 0,C 180,E1 -18541.568,E2 -18541.568} C_VEL
LIN {X 0,Y 256.47,Z 318.519,A -85,B 0,C 180,E1 -18546.716,E2 -18546.716} C_VEL
LIN {X 0,Y 256.435,Z 318.535,A -85,B 0,C 180,E1 -18549.464,E2 -18549.464} C_VEL
LIN {X 0,Y 256.239,Z 318.566,A -85,B 0,C 180,E1 -18554.291,E2 -18554.291} C_VEL
LIN {X 0,Y 256.175,Z 318.571,A -85,B 0,C 180,E1 -18557.564,E2 -18557.564} C_VEL
LIN {X 0,Y 256.148,Z 318.575,A -85,B 0,C 180,E1 -18561.109,E2 -18561.109} C_VEL
LIN {X 0,Y 256.177,Z 318.575,A -85,B 0,C 180,E1 -18565.129,E2 -18565.129} C_VEL
LIN {X 0,Y 256.12,Z 318.577,A -85,B 0,C 180,E1 -18569.599,E2 -18569.599} C_VEL
LIN {X 0,Y 256.074,Z 318.585,A -85,B 0,C 180,E1 -18573.292,E2 -18573.292} C_VEL
LIN {X 0,Y 256.12,Z 318.581,A -85,B 0,C 180,E1 -18577.269,E2 -18577.269} C_VEL
LIN {X 0,Y 256.064,Z 318.583,A -85,B 0,C 180,E1 -18581.201,E2 -18581.201} C_VEL
LIN {X 0,Y 256.05,Z 318.587,A -85,B 0,C 180,E1 -18585.532,E2 -18585.532} C_VEL
LIN {X 0,Y 256.059,Z 318.586,A -85,B 0,C 180,E1 -18588.795,E2 -18588.795} C_VEL
LIN {X 0,Y 256.137,Z 318.577,A -85,B 0,C 180,E1 -18592.866,E2 -18592.866} C_VEL
LIN {X 0,Y 256.072,Z 318.586,A -85,B 0,C 180,E1 -18596.706,E2 -18596.706} C_VEL
LIN {X 0,Y 256.108,Z 318.583,A -85,B 0,C 180,E1 -18600.397,E2 -18600.397} C_VEL
LIN {X 0,Y 256.192,Z 318.571,A -85,B 0,C 180,E1 -18604.86,E2 -18604.86} C_VEL
LIN {X 0,Y 256.222,Z 318.565,A -85,B 0,C 180,E1 -18609.107,E2 -18609.107} C_VEL
LIN {X 0,Y 256.303,Z 318.56,A -85,B 0,C 180,E1 -18614.083,E2 -18614.083} C_VEL
LIN {X 0,Y 256.303,Z 318.71,A -85,B 0,C 180,E1 -18616.439,E2 -18616.439} C_VEL
LIN {X 0,Y 257.408,Z 321.598,A -85,B 0,C 180,E1 -18616.634,E2 -18616.634} C_VEL
LIN {X 0,Y 264.675,Z 340.511,A -85,B 0,C 180,E1 -18617.87,E2 -18617.87} C_VEL
LIN {X 0,Y 267.993,Z 351.008,A -85,B 0,C 180,E1 -18618.463,E2 -18618.463} C_VEL
LIN {X 0,Y 268.191,Z 353.911,A -85,B 0,C 180,E1 -18618.563,E2 -18618.563} C_VEL
LIN {X 0,Y 265.924,Z 426.63,A -85,B 0,C 180,E1 -18620.511,E2 -18620.511} C_VEL
LIN {X 0,Y 265.131,Z 439.961,A -85,B 0,C 180,E1 -18621.183,E2 -18621.183} C_VEL
LIN {X 0,Y 264.169,Z 452.84,A -85,B 0,C 180,E1 -18622.161,E2 -18622.161} C_VEL
LIN {X 0,Y 262.759,Z 465.432,A -85,B 0,C 180,E1 -18623.471,E2 -18623.471} C_VEL
LIN {X 0,Y 261.521,Z 475.492,A -85,B 0,C 180,E1 -18624.818,E2 -18624.818} C_VEL
LIN {X 0,Y 260.015,Z 485.504,A -85,B 0,C 180,E1 -18626.472,E2 -18626.472} C_VEL
LIN {X 0,Y 258.529,Z 495.027,A -85,B 0,C 180,E1 -18628.44,E2 -18628.44} C_VEL
LIN {X 0,Y 257.034,Z 504.065,A -85,B 0,C 180,E1 -18630.781,E2 -18630.781} C_VEL
LIN {X 0,Y 255.916,Z 511.337,A -85,B 0,C 180,E1 -18633.146,E2 -18633.146} C_VEL
LIN {X 0,Y 255.175,Z 517.127,A -85,B 0,C 180,E1 -18635.529,E2 -18635.529} C_VEL
LIN {X 0,Y 254.591,Z 521.694,A -85,B 0,C 180,E1 -18637.931,E2 -18637.931} C_VEL
LIN {X 0,Y 254.261,Z 524.112,A -85,B 0,C 180,E1 -18639.544,E2 -18639.544} C_VEL
LIN {X 0,Y 253.99,Z 526.099,A -85,B 0,C 180,E1 -18641.166,E2 -18641.166} C_VEL
LIN {X 0,Y 253.892,Z 527.638,A -85,B 0,C 180,E1 -18642.792,E2 -18642.792} C_VEL
LIN {X 0,Y 253.845,Z 528.717,A -85,B 0,C 180,E1 -18644.426,E2 -18644.426} C_VEL
LIN {X 0,Y 253.821,Z 529.399,A -85,B 0,C 180,E1 -18646.072,E2 -18646.072} C_VEL
LIN {X 0,Y 253.922,Z 529.68,A -85,B 0,C 180,E1 -18647.723,E2 -18647.723} C_VEL
LIN {X 0,Y 254.312,Z 529.316,A -85,B 0,C 180,E1 -18650.016,E2 -18650.016} C_VEL
LIN {X 0,Y 254.965,Z 527.878,A -85,B 0,C 180,E1 -18652.697,E2 -18652.697} C_VEL
LIN {X 0,Y 255.862,Z 525.707,A -85,B 0,C 180,E1 -18654.982,E2 -18654.982} C_VEL
LIN {X 0,Y 257.244,Z 522.007,A -85,B 0,C 180,E1 -18657.671,E2 -18657.671} C_VEL
LIN {X 0,Y 258.915,Z 517.305,A -85,B 0,C 180,E1 -18660.155,E2 -18660.155} C_VEL
LIN {X 0,Y 260.988,Z 511.274,A -85,B 0,C 180,E1 -18662.583,E2 -18662.583} C_VEL
LIN {X 0,Y 263.503,Z 503.611,A -85,B 0,C 180,E1 -18664.987,E2 -18664.987} C_VEL
LIN {X 0,Y 265.89,Z 495.71,A -85,B 0,C 180,E1 -18666.962,E2 -18666.962} C_VEL
LIN {X 0,Y 268.52,Z 485.982,A -85,B 0,C 180,E1 -18668.911,E2 -18668.911} C_VEL
LIN {X 0,Y 271.215,Z 475.196,A -85,B 0,C 180,E1 -18670.589,E2 -18670.589} C_VEL
LIN {X 0,Y 273.418,Z 464.361,A -85,B 0,C 180,E1 -18671.933,E2 -18671.933} C_VEL
LIN {X 0,Y 275.381,Z 452.68,A -85,B 0,C 180,E1 -18673.05,E2 -18673.05} C_VEL
LIN {X 0,Y 276.855,Z 440.842,A -85,B 0,C 180,E1 -18673.891,E2 -18673.891} C_VEL
LIN {X 0,Y 278.072,Z 427.342,A -85,B 0,C 180,E1 -18674.532,E2 -18674.532} C_VEL
LIN {X 0,Y 280.775,Z 364.801,A -85,B 0,C 180,E1 -18676.16,E2 -18676.16} C_VEL
LIN {X 0,Y 273.986,Z 350.189,A -85,B 0,C 180,E1 -18677.711,E2 -18677.711} C_VEL
LIN {X 0,Y 266.432,Z 336.314,A -85,B 0,C 180,E1 -18679.492,E2 -18679.492} C_VEL
LIN {X 0,Y 261.151,Z 327.628,A -85,B 0,C 180,E1 -18680.798,E2 -18680.798} C_VEL
LIN {X 0,Y 258.215,Z 322.976,A -85,B 0,C 180,E1 -18681.556,E2 -18681.556} C_VEL
LIN {X 0,Y 256.523,Z 320.268,A -85,B 0,C 180,E1 -18682.007,E2 -18682.007} C_VEL
LIN {X 0,Y 256.309,Z 319.616,A -85,B 0,C 180,E1 -18682.156,E2 -18682.156} C_VEL
LIN {X 0,Y 256.106,Z 318.576,A -85,B 0,C 180,E1 -18682.727,E2 -18682.727} C_VEL
LIN {X 0,Y 256.054,Z 318.589,A -85,B 0,C 180,E1 -18686.706,E2 -18686.706} C_VEL
LIN {X 0,Y 256.043,Z 318.592,A -85,B 0,C 180,E1 -18690.392,E2 -18690.392} C_VEL
LIN {X 0,Y 256.12,Z 318.573,A -85,B 0,C 180,E1 -18694.887,E2 -18694.887} C_VEL
LIN {X 0,Y 256.149,Z 318.566,A -85,B 0,C 180,E1 -18699.104,E2 -18699.104} C_VEL
LIN {X 0,Y 256.287,Z 318.55,A -85,B 0,C 180,E1 -18704.085,E2 -18704.085} C_VEL
LIN {X 0,Y 256.284,Z 318.551,A -85,B 0,C 180,E1 -18708.933,E2 -18708.933} C_VEL
LIN {X 0,Y 256.479,Z 318.525,A -85,B 0,C 180,E1 -18712.126,E2 -18712.126} C_VEL
LIN {X 0,Y 256.482,Z 318.529,A -85,B 0,C 180,E1 -18716.859,E2 -18716.859} C_VEL
LIN {X 0,Y 256.752,Z 318.498,A -85,B 0,C 180,E1 -18720,E2 -18720} C_VEL
LIN {X 0,Y 256.703,Z 318.502,A -85,B 0,C 180,E1 -18720.778,E2 -18720.778} C_VEL
LIN {X 0,Y 255.983,Z 318.594,A -85,B 0,C 180,E1 -18722.084,E2 -18722.084} C_VEL
LIN {X 0,Y 253.016,Z 318.963,A -85,B 0,C 180,E1 -18724.208,E2 -18724.208} C_VEL
LIN {X 0,Y 250.537,Z 319.275,A -85,B 0,C 180,E1 -18725.938,E2 -18725.938} C_VEL
LIN {X 0,Y 249.511,Z 319.396,A -85,B 0,C 180,E1 -18727.283,E2 -18727.283} C_VEL
LIN {X 0,Y 249.447,Z 319.398,A -85,B 0,C 180,E1 -18727.739,E2 -18727.739} C_VEL
LIN {X 0,Y 249.241,Z 319.437,A -85,B 0,C 180,E1 -18731.384,E2 -18731.384} C_VEL
LIN {X 0,Y 249.231,Z 319.44,A -85,B 0,C 180,E1 -18736.379,E2 -18736.379} C_VEL
LIN {X 0,Y 249.076,Z 319.459,A -85,B 0,C 180,E1 -18741.519,E2 -18741.519} C_VEL
LIN {X 0,Y 249.121,Z 319.453,A -85,B 0,C 180,E1 -18745.484,E2 -18745.484} C_VEL
LIN {X 0,Y 249.074,Z 319.451,A -85,B 0,C 180,E1 -18748.995,E2 -18748.995} C_VEL
LIN {X 0,Y 249.027,Z 319.456,A -85,B 0,C 180,E1 -18752.427,E2 -18752.427} C_VEL
LIN {X 0,Y 249.067,Z 319.456,A -85,B 0,C 180,E1 -18756.34,E2 -18756.34} C_VEL
LIN {X 0,Y 249.036,Z 319.467,A -85,B 0,C 180,E1 -18760.473,E2 -18760.473} C_VEL
LIN {X 0,Y 249.039,Z 319.461,A -85,B 0,C 180,E1 -18762.804,E2 -18762.804} C_VEL
LIN {X 0,Y 249.058,Z 319.648,A -85,B 0,C 180,E1 -18765.395,E2 -18765.395} C_VEL
LIN {X 0,Y 251.224,Z 326.749,A -85,B 0,C 180,E1 -18769.054,E2 -18769.054} C_VEL
LIN {X 0,Y 253.177,Z 333.829,A -85,B 0,C 180,E1 -18772.348,E2 -18772.348} C_VEL
LIN {X 0,Y 255.554,Z 338.144,A -85,B 0,C 180,E1 -18773.009,E2 -18773.009} C_VEL
LIN {X 0,Y 261.737,Z 349.571,A -85,B 0,C 180,E1 -18774.648,E2 -18774.648} C_VEL
LIN {X 0,Y 268.737,Z 364.013,A -85,B 0,C 180,E1 -18776.408,E2 -18776.408} C_VEL
LIN {X 0,Y 270.79,Z 369.072,A -85,B 0,C 180,E1 -18776.926,E2 -18776.926} C_VEL
LIN {X 0,Y 274.015,Z 389.031,A -85,B 0,C 180,E1 -18778.111,E2 -18778.111} C_VEL
LIN {X 0,Y 272.151,Z 436.315,A -85,B 0,C 180,E1 -18779.361,E2 -18779.361} C_VEL
LIN {X 0,Y 271.222,Z 449.429,A -85,B 0,C 180,E1 -18779.809,E2 -18779.809} C_VEL
LIN {X 0,Y 269.652,Z 462.488,A -85,B 0,C 180,E1 -18780.535,E2 -18780.535} C_VEL
LIN {X 0,Y 267.39,Z 475.454,A -85,B 0,C 180,E1 -18781.553,E2 -18781.553} C_VEL
LIN {X 0,Y 264.979,Z 486.797,A -85,B 0,C 180,E1 -18782.776,E2 -18782.776} C_VEL
LIN {X 0,Y 262.153,Z 498.322,A -85,B 0,C 180,E1 -18784.39,E2 -18784.39} C_VEL
LIN {X 0,Y 259.551,Z 507.639,A -85,B 0,C 180,E1 -18786.039,E2 -18786.039} C_VEL
LIN {X 0,Y 256.825,Z 516.175,A -85,B 0,C 180,E1 -18787.9,E2 -18787.9} C_VEL
LIN {X 0,Y 254.35,Z 523.743,A -85,B 0,C 180,E1 -18789.962,E2 -18789.962} C_VEL
LIN {X 0,Y 252.078,Z 531.216,A -85,B 0,C 180,E1 -18792.562,E2 -18792.562} C_VEL
LIN {X 0,Y 249.84,Z 537.433,A -85,B 0,C 180,E1 -18795.337,E2 -18795.337} C_VEL
LIN {X 0,Y 248.534,Z 541.501,A -85,B 0,C 180,E1 -18797.758,E2 -18797.758} C_VEL
LIN {X 0,Y 247.651,Z 544.543,A -85,B 0,C 180,E1 -18800.199,E2 -18800.199} C_VEL
LIN {X 0,Y 247.264,Z 546.061,A -85,B 0,C 180,E1 -18801.832,E2 -18801.832} C_VEL
LIN {X 0,Y 246.923,Z 547.844,A -85,B 0,C 180,E1 -18805.104,E2 -18805.104} C_VEL
LIN {X 0,Y 246.918,Z 548.163,A -85,B 0,C 180,E1 -18806.739,E2 -18806.739} C_VEL
LIN {X 0,Y 246.996,Z 548.094,A -85,B 0,C 180,E1 -18808.372,E2 -18808.372} C_VEL
LIN {X 0,Y 247.029,Z 547.588,A -85,B 0,C 180,E1 -18810.002,E2 -18810.002} C_VEL
LIN {X 0,Y 247.023,Z 546.679,A -85,B 0,C 180,E1 -18811.633,E2 -18811.633} C_VEL
LIN {X 0,Y 246.994,Z 545.365,A -85,B 0,C 180,E1 -18813.265,E2 -18813.265} C_VEL
LIN {X 0,Y 246.986,Z 543.275,A -85,B 0,C 180,E1 -18815.169,E2 -18815.169} C_VEL
LIN {X 0,Y 247.26,Z 538.695,A -85,B 0,C 180,E1 -18818.173,E2 -18818.173} C_VEL
LIN {X 0,Y 247.728,Z 533.677,A -85,B 0,C 180,E1 -18820.629,E2 -18820.629} C_VEL
LIN {X 0,Y 248.494,Z 527.346,A -85,B 0,C 180,E1 -18823.079,E2 -18823.079} C_VEL
LIN {X 0,Y 249.756,Z 519.41,A -85,B 0,C 180,E1 -18825.507,E2 -18825.507} C_VEL
LIN {X 0,Y 251.091,Z 511.295,A -85,B 0,C 180,E1 -18827.513,E2 -18827.513} C_VEL
LIN {X 0,Y 252.678,Z 501.377,A -85,B 0,C 180,E1 -18829.5,E2 -18829.5} C_VEL
LIN {X 0,Y 253.862,Z 492.926,A -85,B 0,C 180,E1 -18830.884,E2 -18830.884} C_VEL
LIN {X 0,Y 255.598,Z 481.129,A -85,B 0,C 180,E1 -18832.43,E2 -18832.43} C_VEL
LIN {X 0,Y 257.145,Z 468.491,A -85,B 0,C 180,E1 -18833.669,E2 -18833.669} C_VEL
LIN {X 0,Y 258.372,Z 455.121,A -85,B 0,C 180,E1 -18834.617,E2 -18834.617} C_VEL
LIN {X 0,Y 259.158,Z 442.848,A -85,B 0,C 180,E1 -18835.18,E2 -18835.18} C_VEL
LIN {X 0,Y 260.821,Z 386.253,A -85,B 0,C 180,E1 -18836.729,E2 -18836.729} C_VEL
LIN {X 0,Y 256.414,Z 349.51,A -85,B 0,C 180,E1 -18838.219,E2 -18838.219} C_VEL
LIN {X 0,Y 255.338,Z 343.8,A -85,B 0,C 180,E1 -18838.493,E2 -18838.493} C_VEL
LIN {X 0,Y 252.458,Z 335.315,A -85,B 0,C 180,E1 -18839.079,E2 -18839.079} C_VEL
LIN {X 0,Y 249.976,Z 323.559,A -85,B 0,C 180,E1 -18843.324,E2 -18843.324} C_VEL
LIN {X 0,Y 249.064,Z 319.462,A -85,B 0,C 180,E1 -18844.938,E2 -18844.938} C_VEL
LIN {X 0,Y 249.033,Z 319.466,A -85,B 0,C 180,E1 -18848.382,E2 -18848.382} C_VEL
LIN {X 0,Y 249.009,Z 319.469,A -85,B 0,C 180,E1 -18852.792,E2 -18852.792} C_VEL
LIN {X 0,Y 249.017,Z 319.465,A -85,B 0,C 180,E1 -18857.362,E2 -18857.362} C_VEL
LIN {X 0,Y 249.033,Z 319.46,A -85,B 0,C 180,E1 -18861.62,E2 -18861.62} C_VEL
LIN {X 0,Y 249.051,Z 319.456,A -85,B 0,C 180,E1 -18865.64,E2 -18865.64} C_VEL
LIN {X 0,Y 249.06,Z 319.456,A -85,B 0,C 180,E1 -18869.474,E2 -18869.474} C_VEL
